(* IEC 61131-3 sources: mect_apps/AnyTPAC/TestSuite/plc, 74 files *)

(* ---- Crosstable.gvl ---- *)
VAR_GLOBAL
	LogLevel AT %QW0.764:INT;
	Target AT %QD0.768:UDINT;
	Status AT %QD0.772:DINT;
	BUTTON_START AT %QX0.776.0:BOOL;
	BUTTON_STOP AT %QX0.780.0:BOOL;
	BUTTON_RESET AT %QX0.784.0:BOOL;
	Tests AT %QD0.788:UDINT;
	Loops AT %QD0.792:UDINT;
	Errors AT %QD0.796:UDINT;
	Elapsed_s AT %QD0.800:UDINT;
	DisabledTests AT %QW0.804:UINT;
	TestingTests AT %QW0.808:UINT;
	PassedTests AT %QW0.812:UINT;
	FailedTests AT %QW0.816:UINT;
	ETMAX_Task00 AT %QD0.840:UDINT;	(* TSK_GetStatistic().ExecMax *)
	ETMAX_Task01 AT %QD0.844:UDINT;	(* TSK_GetStatistic().ExecMax *)
	ETMAX_Task02 AT %QD0.848:UDINT;	(* TSK_GetStatistic().ExecMax *)
	ETMAX_Task03 AT %QD0.852:UDINT;	(* TSK_GetStatistic().ExecMaxfo *)
	ETMAX_Task04 AT %QD0.856:UDINT;	(* TSK_GetStatistic().ExecMax *)
	ETMAX_Task05 AT %QD0.860:UDINT;	(* TSK_GetStatistic().ExecMax *)
	ETMAX_Task06 AT %QD0.864:UDINT;	(* TSK_GetStatistic().ExecMax *)
	ETMAX_Task07 AT %QD0.868:UDINT;	(* TSK_GetStatistic().ExecMax *)
	ETMAX_Task08 AT %QD0.872:UDINT;	(* TSK_GetStatistic().ExecMax *)
	ETMAX_Task09 AT %QD0.876:UDINT;	(* TSK_GetStatistic().ExecMax *)
	ETMAX_Task10 AT %QD0.880:UDINT;	(* TSK_GetStatistic().ExecMax *)
	ETMAX_Task11 AT %QD0.884:UDINT;	(* TSK_GetStatistic().ExecMax *)
	ETMAX_Task12 AT %QD0.888:UDINT;	(* TSK_GetStatistic().ExecMax *)
	ETMAX_Task13 AT %QD0.892:UDINT;	(* TSK_GetStatistic().ExecMax *)
	ETMAX_Task14 AT %QD0.896:UDINT;	(* TSK_GetStatistic().ExecMaxo *)
	ETMAX_Task15 AT %QD0.900:UDINT;	(* TSK_GetStatistic().ExecMax *)
	ETMAX_Task16 AT %QD0.904:UDINT;	(* TSK_GetStatistic().ExecMax *)
	ETMAX_Task17 AT %QD0.908:UDINT;	(* TSK_GetStatistic().ExecMax *)
	ETMAX_Task18 AT %QD0.912:UDINT;	(* TSK_GetStatistic().ExecMax *)
	ETMAX_Task19 AT %QD0.916:UDINT;	(* TaskInfo *)
	ETAVG_Task00 AT %QD0.960:UDINT;	(* TSK_GetStatistic().ExecAverage *)
	ETAVG_Task01 AT %QD0.964:UDINT;	(* TSK_GetStatistic().ExecAverage *)
	ETAVG_Task02 AT %QD0.968:UDINT;	(* TSK_GetStatistic().ExecAverage *)
	ETAVG_Task03 AT %QD0.972:UDINT;	(* TSK_GetStatistic().ExecAverage *)
	ETAVG_Task04 AT %QD0.976:UDINT;	(* TSK_GetStatistic().ExecAverage *)
	ETAVG_Task05 AT %QD0.980:UDINT;	(* TSK_GetStatistic().ExecAverage *)
	ETAVG_Task06 AT %QD0.984:UDINT;	(* TSK_GetStatistic().ExecAverage *)
	ETAVG_Task07 AT %QD0.988:UDINT;	(* TSK_GetStatistic().ExecAverage *)
	ETAVG_Task08 AT %QD0.992:UDINT;	(* TSK_GetStatistic().ExecAverage *)
	ETAVG_Task09 AT %QD0.996:UDINT;	(* TSK_GetStatistic().ExecAverage *)
	ETAVG_Task10 AT %QD0.1000:UDINT;	(* TSK_GetStatistic().ExecAverage *)
	ETAVG_Task11 AT %QD0.1004:UDINT;	(* TSK_GetStatistic().ExecAverage *)
	ETAVG_Task12 AT %QD0.1008:UDINT;	(* TSK_GetStatistic().ExecAverage *)
	ETAVG_Task13 AT %QD0.1012:UDINT;	(* TSK_GetStatistic().ExecAverage *)
	ETAVG_Task14 AT %QD0.1016:UDINT;	(* TSK_GetStatistic().ExecAverage *)
	ETAVG_Task15 AT %QD0.1020:UDINT;	(* TSK_GetStatistic().ExecAverage *)
	ETAVG_Task16 AT %QD0.1024:UDINT;	(* TSK_GetStatistic().ExecAverage *)
	ETAVG_Task17 AT %QD0.1028:UDINT;	(* TSK_GetStatistic().ExecAverage *)
	ETAVG_Task18 AT %QD0.1032:UDINT;	(* TSK_GetStatistic().ExecAverage *)
	ETAVG_Task19 AT %QD0.1036:UDINT;	(* TSK_GetStatistic().ExecAverage *)
	test_level_01 AT %QW0.1204:UINT;
	test_level_02 AT %QW0.1208:UINT;
	test_level_03 AT %QW0.1212:UINT;
	test_level_04 AT %QW0.1216:UINT;
	test_level_05 AT %QW0.1220:UINT;
	test_level_06 AT %QW0.1224:UINT;
	test_level_07 AT %QW0.1228:UINT;
	test_level_08 AT %QW0.1232:UINT;
	test_level_09 AT %QW0.1236:UINT;
	test_level_10 AT %QW0.1240:UINT;
	test_level_11 AT %QW0.1244:UINT;
	test_level_12 AT %QW0.1248:UINT;
	test_level_13 AT %QW0.1252:UINT;
	test_level_14 AT %QW0.1256:UINT;
	test_level_15 AT %QW0.1260:UINT;
	test_level_16 AT %QW0.1264:UINT;
	test_level_17 AT %QW0.1268:UINT;
	test_level_18 AT %QW0.1272:UINT;
	test_level_19 AT %QW0.1276:UINT;
	test_level_20 AT %QW0.1280:UINT;
	test_level_21 AT %QW0.1284:UINT;
	test_level_22 AT %QW0.1288:UINT;
	test_level_23 AT %QW0.1292:UINT;
	test_level_24 AT %QW0.1296:UINT;
	test_level_25 AT %QW0.1300:UINT;
	test_level_26 AT %QW0.1304:UINT;
	test_level_27 AT %QW0.1308:UINT;
	test_level_28 AT %QW0.1312:UINT;
	test_level_29 AT %QW0.1316:UINT;
	test_level_30 AT %QW0.1320:UINT;
	test_level_31 AT %QW0.1324:UINT;
	test_level_32 AT %QW0.1328:UINT;
	test_level_33 AT %QW0.1332:UINT;
	test_level_34 AT %QW0.1336:UINT;
	test_level_35 AT %QW0.1340:UINT;
	test_level_36 AT %QW0.1344:UINT;
	test_level_37 AT %QW0.1348:UINT;
	test_level_38 AT %QW0.1352:UINT;
	test_level_39 AT %QW0.1356:UINT;
	test_level_40 AT %QW0.1360:UINT;
	test_level_41 AT %QW0.1364:UINT;
	test_level_42 AT %QW0.1368:UINT;
	test_level_43 AT %QW0.1372:UINT;
	test_level_44 AT %QW0.1376:UINT;
	test_level_45 AT %QW0.1380:UINT;
	test_level_46 AT %QW0.1384:UINT;
	test_level_47 AT %QW0.1388:UINT;
	test_level_48 AT %QW0.1392:UINT;
	test_level_49 AT %QW0.1396:UINT;
	test_level_50 AT %QW0.1400:UINT;
	test_level_51 AT %QW0.1404:UINT;
	test_level_52 AT %QW0.1408:UINT;
	test_level_53 AT %QW0.1412:UINT;
	test_level_54 AT %QW0.1416:UINT;
	test_level_55 AT %QW0.1420:UINT;
	test_level_56 AT %QW0.1424:UINT;
	test_level_57 AT %QW0.1428:UINT;
	test_level_58 AT %QW0.1432:UINT;
	test_level_59 AT %QW0.1436:UINT;
	test_level_60 AT %QW0.1440:UINT;
	test_counter_01 AT %QD0.1604:UDINT;
	test_counter_02 AT %QD0.1608:UDINT;
	test_counter_03 AT %QD0.1612:UDINT;
	test_counter_04 AT %QD0.1616:UDINT;
	test_counter_05 AT %QD0.1620:UDINT;
	test_counter_06 AT %QD0.1624:UDINT;
	test_counter_07 AT %QD0.1628:UDINT;
	test_counter_08 AT %QD0.1632:UDINT;
	test_counter_09 AT %QD0.1636:UDINT;
	test_counter_10 AT %QD0.1640:UDINT;
	test_counter_11 AT %QD0.1644:UDINT;
	test_counter_12 AT %QD0.1648:UDINT;
	test_counter_13 AT %QD0.1652:UDINT;
	test_counter_14 AT %QD0.1656:UDINT;
	test_counter_15 AT %QD0.1660:UDINT;
	test_counter_16 AT %QD0.1664:UDINT;
	test_counter_17 AT %QD0.1668:UDINT;
	test_counter_18 AT %QD0.1672:UDINT;
	test_counter_19 AT %QD0.1676:UDINT;
	test_counter_20 AT %QD0.1680:UDINT;
	test_counter_21 AT %QD0.1684:UDINT;
	test_counter_22 AT %QD0.1688:UDINT;
	test_counter_23 AT %QD0.1692:UDINT;
	test_counter_24 AT %QD0.1696:UDINT;
	test_counter_25 AT %QD0.1700:UDINT;
	test_counter_26 AT %QD0.1704:UDINT;
	test_counter_27 AT %QD0.1708:UDINT;
	test_counter_28 AT %QD0.1712:UDINT;
	test_counter_29 AT %QD0.1716:UDINT;
	test_counter_30 AT %QD0.1720:UDINT;
	test_counter_31 AT %QD0.1724:UDINT;
	test_counter_32 AT %QD0.1728:UDINT;
	test_counter_33 AT %QD0.1732:UDINT;
	test_counter_34 AT %QD0.1736:UDINT;
	test_counter_35 AT %QD0.1740:UDINT;
	test_counter_36 AT %QD0.1744:UDINT;
	test_counter_37 AT %QD0.1748:UDINT;
	test_counter_38 AT %QD0.1752:UDINT;
	test_counter_39 AT %QD0.1756:UDINT;
	test_counter_40 AT %QD0.1760:UDINT;
	test_counter_41 AT %QD0.1764:UDINT;
	test_counter_42 AT %QD0.1768:UDINT;
	test_counter_43 AT %QD0.1772:UDINT;
	test_counter_44 AT %QD0.1776:UDINT;
	test_counter_45 AT %QD0.1780:UDINT;
	test_counter_46 AT %QD0.1784:UDINT;
	test_counter_47 AT %QD0.1788:UDINT;
	test_counter_48 AT %QD0.1792:UDINT;
	test_counter_49 AT %QD0.1796:UDINT;
	test_counter_50 AT %QD0.1800:UDINT;
	test_counter_51 AT %QD0.1804:UDINT;
	test_counter_52 AT %QD0.1808:UDINT;
	test_counter_53 AT %QD0.1812:UDINT;
	test_counter_54 AT %QD0.1816:UDINT;
	test_counter_55 AT %QD0.1820:UDINT;
	test_counter_56 AT %QD0.1824:UDINT;
	test_counter_57 AT %QD0.1828:UDINT;
	test_counter_58 AT %QD0.1832:UDINT;
	test_counter_59 AT %QD0.1836:UDINT;
	test_counter_60 AT %QD0.1840:UDINT;
	test_loops_01 AT %QD0.2004:UDINT;
	test_loops_02 AT %QD0.2008:UDINT;
	test_loops_03 AT %QD0.2012:UDINT;
	test_loops_04 AT %QD0.2016:UDINT;
	test_loops_05 AT %QD0.2020:UDINT;
	test_loops_06 AT %QD0.2024:UDINT;
	test_loops_07 AT %QD0.2028:UDINT;
	test_loops_08 AT %QD0.2032:UDINT;
	test_loops_09 AT %QD0.2036:UDINT;
	test_loops_10 AT %QD0.2040:UDINT;
	test_loops_11 AT %QD0.2044:UDINT;
	test_loops_12 AT %QD0.2048:UDINT;
	test_loops_13 AT %QD0.2052:UDINT;
	test_loops_14 AT %QD0.2056:UDINT;
	test_loops_15 AT %QD0.2060:UDINT;
	test_loops_16 AT %QD0.2064:UDINT;
	test_loops_17 AT %QD0.2068:UDINT;
	test_loops_18 AT %QD0.2072:UDINT;
	test_loops_19 AT %QD0.2076:UDINT;
	test_loops_20 AT %QD0.2080:UDINT;
	test_loops_21 AT %QD0.2084:UDINT;
	test_loops_22 AT %QD0.2088:UDINT;
	test_loops_23 AT %QD0.2092:UDINT;
	test_loops_24 AT %QD0.2096:UDINT;
	test_loops_25 AT %QD0.2100:UDINT;
	test_loops_26 AT %QD0.2104:UDINT;
	test_loops_27 AT %QD0.2108:UDINT;
	test_loops_28 AT %QD0.2112:UDINT;
	test_loops_29 AT %QD0.2116:UDINT;
	test_loops_30 AT %QD0.2120:UDINT;
	test_loops_31 AT %QD0.2124:UDINT;
	test_loops_32 AT %QD0.2128:UDINT;
	test_loops_33 AT %QD0.2132:UDINT;
	test_loops_34 AT %QD0.2136:UDINT;
	test_loops_35 AT %QD0.2140:UDINT;
	test_loops_36 AT %QD0.2144:UDINT;
	test_loops_37 AT %QD0.2148:UDINT;
	test_loops_38 AT %QD0.2152:UDINT;
	test_loops_39 AT %QD0.2156:UDINT;
	test_loops_40 AT %QD0.2160:UDINT;
	test_loops_41 AT %QD0.2164:UDINT;
	test_loops_42 AT %QD0.2168:UDINT;
	test_loops_43 AT %QD0.2172:UDINT;
	test_loops_44 AT %QD0.2176:UDINT;
	test_loops_45 AT %QD0.2180:UDINT;
	test_loops_46 AT %QD0.2184:UDINT;
	test_loops_47 AT %QD0.2188:UDINT;
	test_loops_48 AT %QD0.2192:UDINT;
	test_loops_49 AT %QD0.2196:UDINT;
	test_loops_50 AT %QD0.2200:UDINT;
	test_loops_51 AT %QD0.2204:UDINT;
	test_loops_52 AT %QD0.2208:UDINT;
	test_loops_53 AT %QD0.2212:UDINT;
	test_loops_54 AT %QD0.2216:UDINT;
	test_loops_55 AT %QD0.2220:UDINT;
	test_loops_56 AT %QD0.2224:UDINT;
	test_loops_57 AT %QD0.2228:UDINT;
	test_loops_58 AT %QD0.2232:UDINT;
	test_loops_59 AT %QD0.2236:UDINT;
	test_loops_60 AT %QD0.2240:UDINT;
	test_errors_01 AT %QD0.2404:UDINT;
	test_errors_02 AT %QD0.2408:UDINT;
	test_errors_03 AT %QD0.2412:UDINT;
	test_errors_04 AT %QD0.2416:UDINT;
	test_errors_05 AT %QD0.2420:UDINT;
	test_errors_06 AT %QD0.2424:UDINT;
	test_errors_07 AT %QD0.2428:UDINT;
	test_errors_08 AT %QD0.2432:UDINT;
	test_errors_09 AT %QD0.2436:UDINT;
	test_errors_10 AT %QD0.2440:UDINT;
	test_errors_11 AT %QD0.2444:UDINT;
	test_errors_12 AT %QD0.2448:UDINT;
	test_errors_13 AT %QD0.2452:UDINT;
	test_errors_14 AT %QD0.2456:UDINT;
	test_errors_15 AT %QD0.2460:UDINT;
	test_errors_16 AT %QD0.2464:UDINT;
	test_errors_17 AT %QD0.2468:UDINT;
	test_errors_18 AT %QD0.2472:UDINT;
	test_errors_19 AT %QD0.2476:UDINT;
	test_errors_20 AT %QD0.2480:UDINT;
	test_errors_21 AT %QD0.2484:UDINT;
	test_errors_22 AT %QD0.2488:UDINT;
	test_errors_23 AT %QD0.2492:UDINT;
	test_errors_24 AT %QD0.2496:UDINT;
	test_errors_25 AT %QD0.2500:UDINT;
	test_errors_26 AT %QD0.2504:UDINT;
	test_errors_27 AT %QD0.2508:UDINT;
	test_errors_28 AT %QD0.2512:UDINT;
	test_errors_29 AT %QD0.2516:UDINT;
	test_errors_30 AT %QD0.2520:UDINT;
	test_errors_31 AT %QD0.2524:UDINT;
	test_errors_32 AT %QD0.2528:UDINT;
	test_errors_33 AT %QD0.2532:UDINT;
	test_errors_34 AT %QD0.2536:UDINT;
	test_errors_35 AT %QD0.2540:UDINT;
	test_errors_36 AT %QD0.2544:UDINT;
	test_errors_37 AT %QD0.2548:UDINT;
	test_errors_38 AT %QD0.2552:UDINT;
	test_errors_39 AT %QD0.2556:UDINT;
	test_errors_40 AT %QD0.2560:UDINT;
	test_errors_41 AT %QD0.2564:UDINT;
	test_errors_42 AT %QD0.2568:UDINT;
	test_errors_43 AT %QD0.2572:UDINT;
	test_errors_44 AT %QD0.2576:UDINT;
	test_errors_45 AT %QD0.2580:UDINT;
	test_errors_46 AT %QD0.2584:UDINT;
	test_errors_47 AT %QD0.2588:UDINT;
	test_errors_48 AT %QD0.2592:UDINT;
	test_errors_49 AT %QD0.2596:UDINT;
	test_errors_50 AT %QD0.2600:UDINT;
	test_errors_51 AT %QD0.2604:UDINT;
	test_errors_52 AT %QD0.2608:UDINT;
	test_errors_53 AT %QD0.2612:UDINT;
	test_errors_54 AT %QD0.2616:UDINT;
	test_errors_55 AT %QD0.2620:UDINT;
	test_errors_56 AT %QD0.2624:UDINT;
	test_errors_57 AT %QD0.2628:UDINT;
	test_errors_58 AT %QD0.2632:UDINT;
	test_errors_59 AT %QD0.2636:UDINT;
	test_errors_60 AT %QD0.2640:UDINT;
	RTU0_TYPE_PORT AT %ID0.20000:UDINT;
	RTU0_BAUDRATE AT %ID0.20004:UDINT;
	RTU0_STATUS AT %ID0.20008:UDINT;
	RTU0_READS AT %ID0.20012:UDINT;
	RTU0_WRITES AT %ID0.20016:UDINT;
	RTU0_TIMEOUTS AT %ID0.20020:UDINT;
	RTU0_COMM_ERRORS AT %ID0.20024:UDINT;
	RTU0_LAST_ERROR AT %ID0.20028:UDINT;
	RTU0_WRITE_QUEUE AT %ID0.20032:UDINT;
	RTU0_BUS_LOAD AT %ID0.20036:UDINT;
	RTU1_TYPE_PORT AT %ID0.20040:UDINT;
	RTU1_BAUDRATE AT %ID0.20044:UDINT;
	RTU1_STATUS AT %ID0.20048:UDINT;
	RTU1_READS AT %ID0.20052:UDINT;
	RTU1_WRITES AT %ID0.20056:UDINT;
	RTU1_TIMEOUTS AT %ID0.20060:UDINT;
	RTU1_COMM_ERRORS AT %ID0.20064:UDINT;
	RTU1_LAST_ERROR AT %ID0.20068:UDINT;
	RTU1_WRITE_QUEUE AT %ID0.20072:UDINT;
	RTU1_BUS_LOAD AT %ID0.20076:UDINT;
	RTU3_TYPE_PORT AT %ID0.20080:UDINT;
	RTU3_BAUDRATE AT %ID0.20084:UDINT;
	RTU3_STATUS AT %ID0.20088:UDINT;
	RTU3_READS AT %ID0.20092:UDINT;
	RTU3_WRITES AT %ID0.20096:UDINT;
	RTU3_TIMEOUTS AT %ID0.20100:UDINT;
	RTU3_COMM_ERRORS AT %ID0.20104:UDINT;
	RTU3_LAST_ERROR AT %ID0.20108:UDINT;
	RTU3_WRITE_QUEUE AT %ID0.20112:UDINT;
	RTU3_BUS_LOAD AT %ID0.20116:UDINT;
	CAN0_TYPE_PORT AT %ID0.20120:UDINT;
	CAN0_BAUDRATE AT %ID0.20124:UDINT;
	CAN0_STATUS AT %ID0.20128:UDINT;
	CAN0_READS AT %ID0.20132:UDINT;
	CAN0_WRITES AT %ID0.20136:UDINT;
	CAN0_TIMEOUTS AT %ID0.20140:UDINT;
	CAN0_COMM_ERRORS AT %ID0.20144:UDINT;
	CAN0_LAST_ERROR AT %ID0.20148:UDINT;
	CAN0_WRITE_QUEUE AT %ID0.20152:UDINT;
	CAN0_BUS_LOAD AT %ID0.20156:UDINT;
	CAN1_TYPE_PORT AT %ID0.20160:UDINT;
	CAN1_BAUDRATE AT %ID0.20164:UDINT;
	CAN1_STATUS AT %ID0.20168:UDINT;
	CAN1_READS AT %ID0.20172:UDINT;
	CAN1_WRITES AT %ID0.20176:UDINT;
	CAN1_TIMEOUTS AT %ID0.20180:UDINT;
	CAN1_COMM_ERRORS AT %ID0.20184:UDINT;
	CAN1_LAST_ERROR AT %ID0.20188:UDINT;
	CAN1_WRITE_QUEUE AT %ID0.20192:UDINT;
	CAN1_BUS_LOAD AT %ID0.20196:UDINT;
	TCPS_TYPE_PORT AT %ID0.20200:UDINT;
	TCPS_IP_ADDRESS AT %ID0.20204:UDINT;
	TCPS_STATUS AT %ID0.20208:UDINT;
	TCPS_READS AT %ID0.20212:UDINT;
	TCPS_WRITES AT %ID0.20216:UDINT;
	TCPS_TIMEOUTS AT %ID0.20220:UDINT;
	TCPS_COMM_ERRORS AT %ID0.20224:UDINT;
	TCPS_LAST_ERROR AT %ID0.20228:UDINT;
	TCPS_WRITE_QUEUE AT %ID0.20232:UDINT;
	TCPS_BUS_LOAD AT %ID0.20236:UDINT;
	TCP0_TYPE_PORT AT %ID0.20240:UDINT;
	TCP0_IP_ADDRESS AT %ID0.20244:UDINT;
	TCP0_STATUS AT %ID0.20248:UDINT;
	TCP0_READS AT %ID0.20252:UDINT;
	TCP0_WRITES AT %ID0.20256:UDINT;
	TCP0_TIMEOUTS AT %ID0.20260:UDINT;
	TCP0_COMM_ERRORS AT %ID0.20264:UDINT;
	TCP0_LAST_ERROR AT %ID0.20268:UDINT;
	TCP0_WRITE_QUEUE AT %ID0.20272:UDINT;
	TCP0_BUS_LOAD AT %ID0.20276:UDINT;
	TCP1_TYPE_PORT AT %ID0.20280:UDINT;
	TCP1_IP_ADDRESS AT %ID0.20284:UDINT;
	TCP1_STATUS AT %ID0.20288:UDINT;
	TCP1_READS AT %ID0.20292:UDINT;
	TCP1_WRITES AT %ID0.20296:UDINT;
	TCP1_TIMEOUTS AT %ID0.20300:UDINT;
	TCP1_COMM_ERRORS AT %ID0.20304:UDINT;
	TCP1_LAST_ERROR AT %ID0.20308:UDINT;
	TCP1_WRITE_QUEUE AT %ID0.20312:UDINT;
	TCP1_BUS_LOAD AT %ID0.20316:UDINT;
	TCP2_TYPE_PORT AT %ID0.20320:UDINT;
	TCP2_IP_ADDRESS AT %ID0.20324:UDINT;
	TCP2_STATUS AT %ID0.20328:UDINT;
	TCP2_READS AT %ID0.20332:UDINT;
	TCP2_WRITES AT %ID0.20336:UDINT;
	TCP2_TIMEOUTS AT %ID0.20340:UDINT;
	TCP2_COMM_ERRORS AT %ID0.20344:UDINT;
	TCP2_LAST_ERROR AT %ID0.20348:UDINT;
	TCP2_WRITE_QUEUE AT %ID0.20352:UDINT;
	TCP2_BUS_LOAD AT %ID0.20356:UDINT;
	TCP3_TYPE_PORT AT %ID0.20360:UDINT;
	TCP3_IP_ADDRESS AT %ID0.20364:UDINT;
	TCP3_STATUS AT %ID0.20368:UDINT;
	TCP3_READS AT %ID0.20372:UDINT;
	TCP3_WRITES AT %ID0.20376:UDINT;
	TCP3_TIMEOUTS AT %ID0.20380:UDINT;
	TCP3_COMM_ERRORS AT %ID0.20384:UDINT;
	TCP3_LAST_ERROR AT %ID0.20388:UDINT;
	TCP3_WRITE_QUEUE AT %ID0.20392:UDINT;
	TCP3_BUS_LOAD AT %ID0.20396:UDINT;
	TCP4_TYPE_PORT AT %ID0.20400:UDINT;
	TCP4_IP_ADDRESS AT %ID0.20404:UDINT;
	TCP4_STATUS AT %ID0.20408:UDINT;
	TCP4_READS AT %ID0.20412:UDINT;
	TCP4_WRITES AT %ID0.20416:UDINT;
	TCP4_TIMEOUTS AT %ID0.20420:UDINT;
	TCP4_COMM_ERRORS AT %ID0.20424:UDINT;
	TCP4_LAST_ERROR AT %ID0.20428:UDINT;
	TCP4_WRITE_QUEUE AT %ID0.20432:UDINT;
	TCP4_BUS_LOAD AT %ID0.20436:UDINT;
	TCP5_TYPE_PORT AT %ID0.20440:UDINT;
	TCP5_IP_ADDRESS AT %ID0.20444:UDINT;
	TCP5_STATUS AT %ID0.20448:UDINT;
	TCP5_READS AT %ID0.20452:UDINT;
	TCP5_WRITES AT %ID0.20456:UDINT;
	TCP5_TIMEOUTS AT %ID0.20460:UDINT;
	TCP5_COMM_ERRORS AT %ID0.20464:UDINT;
	TCP5_LAST_ERROR AT %ID0.20468:UDINT;
	TCP5_WRITE_QUEUE AT %ID0.20472:UDINT;
	TCP5_BUS_LOAD AT %ID0.20476:UDINT;
	TCP6_TYPE_PORT AT %ID0.20480:UDINT;
	TCP6_IP_ADDRESS AT %ID0.20484:UDINT;
	TCP6_STATUS AT %ID0.20488:UDINT;
	TCP6_READS AT %ID0.20492:UDINT;
	TCP6_WRITES AT %ID0.20496:UDINT;
	TCP6_TIMEOUTS AT %ID0.20500:UDINT;
	TCP6_COMM_ERRORS AT %ID0.20504:UDINT;
	TCP6_LAST_ERROR AT %ID0.20508:UDINT;
	TCP6_WRITE_QUEUE AT %ID0.20512:UDINT;
	TCP6_BUS_LOAD AT %ID0.20516:UDINT;
	TCP7_TYPE_PORT AT %ID0.20520:UDINT;
	TCP7_IP_ADDRESS AT %ID0.20524:UDINT;
	TCP7_STATUS AT %ID0.20528:UDINT;
	TCP7_READS AT %ID0.20532:UDINT;
	TCP7_WRITES AT %ID0.20536:UDINT;
	TCP7_TIMEOUTS AT %ID0.20540:UDINT;
	TCP7_COMM_ERRORS AT %ID0.20544:UDINT;
	TCP7_LAST_ERROR AT %ID0.20548:UDINT;
	TCP7_WRITE_QUEUE AT %ID0.20552:UDINT;
	TCP7_BUS_LOAD AT %ID0.20556:UDINT;
	TCP8_TYPE_PORT AT %ID0.20560:UDINT;
	TCP8_IP_ADDRESS AT %ID0.20564:UDINT;
	TCP8_STATUS AT %ID0.20568:UDINT;
	TCP8_READS AT %ID0.20572:UDINT;
	TCP8_WRITES AT %ID0.20576:UDINT;
	TCP8_TIMEOUTS AT %ID0.20580:UDINT;
	TCP8_COMM_ERRORS AT %ID0.20584:UDINT;
	TCP8_LAST_ERROR AT %ID0.20588:UDINT;
	TCP8_WRITE_QUEUE AT %ID0.20592:UDINT;
	TCP8_BUS_LOAD AT %ID0.20596:UDINT;
	TCP9_TYPE_PORT AT %ID0.20600:UDINT;
	TCP9_IP_ADDRESS AT %ID0.20604:UDINT;
	TCP9_STATUS AT %ID0.20608:UDINT;
	TCP9_READS AT %ID0.20612:UDINT;
	TCP9_WRITES AT %ID0.20616:UDINT;
	TCP9_TIMEOUTS AT %ID0.20620:UDINT;
	TCP9_COMM_ERRORS AT %ID0.20624:UDINT;
	TCP9_LAST_ERROR AT %ID0.20628:UDINT;
	TCP9_WRITE_QUEUE AT %ID0.20632:UDINT;
	TCP9_BUS_LOAD AT %ID0.20636:UDINT;
	NODE_01_DEV_NODE AT %ID0.20688:UDINT;
	NODE_01_STATUS AT %ID0.20692:UDINT;
	NODE_02_DEV_NODE AT %ID0.20696:UDINT;
	NODE_02_STATUS AT %ID0.20700:UDINT;
	NODE_03_DEV_NODE AT %ID0.20704:UDINT;
	NODE_03_STATUS AT %ID0.20708:UDINT;
	NODE_04_DEV_NODE AT %ID0.20712:UDINT;
	NODE_04_STATUS AT %ID0.20716:UDINT;
	NODE_05_DEV_NODE AT %ID0.20720:UDINT;
	NODE_05_STATUS AT %ID0.20724:UDINT;
	NODE_06_DEV_NODE AT %ID0.20728:UDINT;
	NODE_06_STATUS AT %ID0.20732:UDINT;
	NODE_07_DEV_NODE AT %ID0.20736:UDINT;
	NODE_07_STATUS AT %ID0.20740:UDINT;
	NODE_08_DEV_NODE AT %ID0.20744:UDINT;
	NODE_08_STATUS AT %ID0.20748:UDINT;
	NODE_09_DEV_NODE AT %ID0.20752:UDINT;
	NODE_09_STATUS AT %ID0.20756:UDINT;
	NODE_10_DEV_NODE AT %ID0.20760:UDINT;
	NODE_10_STATUS AT %ID0.20764:UDINT;
	NODE_11_DEV_NODE AT %ID0.20768:UDINT;
	NODE_11_STATUS AT %ID0.20772:UDINT;
	NODE_12_DEV_NODE AT %ID0.20776:UDINT;
	NODE_12_STATUS AT %ID0.20780:UDINT;
	NODE_13_DEV_NODE AT %ID0.20784:UDINT;
	NODE_13_STATUS AT %ID0.20788:UDINT;
	NODE_14_DEV_NODE AT %ID0.20792:UDINT;
	NODE_14_STATUS AT %ID0.20796:UDINT;
	NODE_15_DEV_NODE AT %ID0.20800:UDINT;
	NODE_15_STATUS AT %ID0.20804:UDINT;
	NODE_16_DEV_NODE AT %ID0.20808:UDINT;
	NODE_16_STATUS AT %ID0.20812:UDINT;
	PLC_time AT %ID0.21560:REAL;	(* Seconds since boot (reset each 24h) *)
	PLC_timeMin AT %ID0.21564:REAL;	(* 10 seconds window start *)
	PLC_timeMax AT %ID0.21568:REAL;	(* 10 seconds window stop *)
	PLC_timeWin AT %QD0.21572:REAL;	(* Graph display window *)
	PLC_Version AT %IW0.21576:UINT;	(* Run Time version *)
	PLC_EngineStatus AT %IW0.21580:UINT;	(* PLC status *)
	PLC_ResetValues AT %QX0.21584.0:BOOL;	(* Diagnostic variables reset *)
	PLC_buzzerOn AT %QX0.21588.0:BOOL;	(* Buzzer sound (enable = 1 disable = 0) *)
	PLC_PLC_Version AT %QW0.21592:UINT;	(* PLC application version *)
	PLC_HMI_Version AT %QW0.21596:UINT;	(* HMI application version *)
	PLC_Year AT %IW0.21640:UINT;	(* Currently year *)
	PLC_Month AT %IW0.21644:UINT;	(* Currently month *)
	PLC_Day AT %IW0.21648:UINT;	(* Currently day *)
	PLC_Hours AT %IW0.21652:UINT;	(* Currently hour *)
	PLC_Minutes AT %IW0.21656:UINT;	(* Currently minutes *)
	PLC_Seconds AT %IW0.21660:UINT;	(* Currently seconds *)
	PLC_UPTIME_s AT %ID0.21664:UDINT;	(* Uptime in seconds (wraps in 136 years) *)
	PLC_UPTIME_cs AT %ID0.21668:UDINT;	(* Uptime in centiseconds = 10 ms (wraps in 497 days) *)
	PLC_WATCHDOGEN AT %QX0.21672.0:BOOL;	(* Enable Watchdog *)
	PLC_WATCHDOG_ms AT %QD0.21676:UDINT;	(* Reset Watchdog timer *)
	PLC_PRODUCT_ID AT %ID0.21680:UDINT;	(* TP/TPAC/TPLC Product ID (Hex) *)
	PLC_SERIAL_NUMBER AT %ID0.21684:UDINT;	(* TP/TPAC/TPLC Serial Number *)
	PLC_HMI_PAGE AT %QD0.21688:DINT;	(* HMI Page (page100=0x00000100) *)
	PLC_BEEP_VOLUME AT %QB0.21740:BYTE;	(* Beep volume (when buzzerOn) *)
	PLC_TOUCH_VOLUME AT %QB0.21744:BYTE;	(* Touch volume *)
	PLC_ALARM_VOLUME AT %QB0.21748:BYTE;	(* Alarm volume (when alarm) *)
	PLC_BUZZER AT %QD0.21752:UDINT;	(* Enable dynamic buzzer sound (0x44332211 up=0x11(%) on=0x22(cs) off=0x33(cs) rep=0x44(times)) *)
END_VAR

(* ---- Resource1.gvl ---- *)
(* Global variable file *)

VAR_GLOBAL

	log_file : F_SYNC_FILE;

	test_names : array [1..test_num] of string := [
	(* 01 *) 'ATCM_IEC1131_3:bool_to_*',
	(* 02 *) 'ATCM_IEC1131_3:byte_to_*',
	(* 03 *) 'ATCM_IEC1131_3:dint_to_*',
	(* 04 *) 'ATCM_IEC1131_3:dword_to_*',
	(* 05 *) 'ATCM_IEC1131_3:int_to_*',
	(* 06 *) 'ATCM_IEC1131_3:lreal_to_*',
	(* 07 *) 'ATCM_IEC1131_3:real_to_*',
	(* 08 *) 'ATCM_IEC1131_3:string_to_*',
	(* 09 *) 'ATCM_IEC1131_3:time_to_*',
	(* 10 *) 'ATCM_IEC1131_3:trunc_to_*',
	(* 11 *) 'ATCM_IEC1131_3:udint_to_*',
	(* 12 *) 'ATCM_IEC1131_3:uint_to_*',
	(* 13 *) 'ATCM_IEC1131_3:word_to_*',
	(* 14 *) 'ATCM_IEC1131_3:ABS',
	(* 15 *) 'ATCM_IEC1131_3:TRIG_INV=ASIN+ACOS+ATAN',
	(* 16 *) 'ATCM_IEC1131_3:TRIG=SIN+COS+TAN',
	(* 17 *) 'ATCM_IEC1131_3:POW=EXP+LN+LOG+SQRT',
	(* 18 *) 'ATCM_IEC1131_3:ADD',
	(* 19 *) 'ATCM_IEC1131_3:DIV',
	(* 20 *) 'ATCM_IEC1131_3:EXPT',
	(* 21 *) 'ATCM_IEC1131_3:MOD',
	(* 22 *) 'ATCM_IEC1131_3:MOVE',
	(* 23 *) 'ATCM_IEC1131_3:MUL',
	(* 24 *) 'ATCM_IEC1131_3:SUB',
	(* 25 *) 'ATCM_IEC1131_3:RO=ROL+ROR',
	(* 26 *) 'ATCM_IEC1131_3:SH=SHL+SHR',
	(* 27 *) 'ATCM_IEC1131_3:AND',
	(* 28 *) 'ATCM_IEC1131_3:NOT',
	(* 29 *) 'ATCM_IEC1131_3:OR',
	(* 30 *) 'ATCM_IEC1131_3:XOR',
	(* 31 *) 'ATCM_IEC1131_3:LIMIT',
	(* 32 *) 'ATCM_IEC1131_3:MAX',
	(* 33 *) 'ATCM_IEC1131_3:MIN',
	(* 34 *) 'ATCM_IEC1131_3:MUX',
	(* 35 *) 'ATCM_IEC1131_3:SEL',
	(* 36 *) 'ATCM_IEC1131_3:EQ',
	(* 37 *) 'ATCM_IEC1131_3:GE',
	(* 38 *) 'ATCM_IEC1131_3:GT',
	(* 39 *) 'ATCM_IEC1131_3:LE',
	(* 40 *) 'ATCM_IEC1131_3:LT',
	(* 41 *) 'ATCM_IEC1131_3:NE',
	(* 42 *) 'ATCM_IEC1131_3:CONCAT',
	(* 43 *) 'ATCM_IEC1131_3:DELETE',
	(* 44 *) 'ATCM_IEC1131_3:FIND',
	(* 45 *) 'ATCM_IEC1131_3:INSERT',
	(* 46 *) 'ATCM_IEC1131_3:LEFT=LEFT+RIGHT',
	(* 47 *) 'ATCM_IEC1131_3:LEN',
	(* 48 *) 'ATCM_IEC1131_3:MID',
	(* 49 *) 'ATCM_IEC1131_3:REPLACE',
	(* 50 *) 'ATCM_IEC1131_3:ADDTIME+SUBTIME',
	(* 51 *) 'ATCM_IEC1131_3:DIVTIME+MULTIME',
	(* 52 *) 'ATCM_IEC1131_3:RS+SR',
	(* 53 *) 'ATCM_IEC1131_3:F_TRIG+R_TRIG',
	(* 54 *) 'ATCM_IEC1131_3:CTD+CTU+CTUD',
	(* 55 *) 'ATCM_IEC1131_3:TOF+TON+TP',
	(* 56 *) 'ATCM_Utility:BYTE_SWAP_DWORD+WORD',
	(* 57 *) 'ATCM_Utility:COPY_FROM+TO_BYTE_ARRAY',
	(* 58 *) 'ATCM_Utility:HI+LO_BYTE+WORD',
	(* 59 *) 'ATCM_Utility:MAKE_DWORD+WORD',
    (* 60 *) ''
	];

END_VAR

(* ---- ResetCounters.st ---- *)
(*[[
]]*)
FUNCTION ResetCounters
#import "Crosstable.gvl"
#import "Resource1.gvl"
VAR
	retval : WORD;
END_VAR;

	Elapsed_s := 0;
	Loops := 0;
	Errors := 0;

	(* no Task00_TestInit *)
	retval := TSK_ClearStatistic('Task01_TestManager');
	retval := TSK_ClearStatistic('Task02_TestMonitor');

	retval := TSK_ClearStatistic('Task03_ATCM_File');
	retval := TSK_ClearStatistic('Task04_ATCM_IEC1131_3_A');
	retval := TSK_ClearStatistic('Task05_ATCM_IEC1131_3_B');
	retval := TSK_ClearStatistic('Task06_ATCM_IEC1131_3_C');
	retval := TSK_ClearStatistic('Task07_ATCM_IEC1131_3_D');
	retval := TSK_ClearStatistic('Task08_ATCM_IEC1131_3_E');
	retval := TSK_ClearStatistic('Task09_ATCM_IEC1131_3_F');
	retval := TSK_ClearStatistic('Task10_ATCM_IEC1131_3_G');
	retval := TSK_ClearStatistic('Task11_ATCM_IEC1131_3_H');
	retval := TSK_ClearStatistic('Task12_ATCM_IEC1131_3_I');
	retval := TSK_ClearStatistic('Task13_ATCM_IEC1131_3_J');
	retval := TSK_ClearStatistic('Task14_ATCM_IEC1131_3_K');
	retval := TSK_ClearStatistic('Task15_ATCM_IEC1131_3_L');
	retval := TSK_ClearStatistic('Task16_ATCM_IEC1131_3_M');
	retval := TSK_ClearStatistic('Task17_ATCM_System');
	retval := TSK_ClearStatistic('Task18_ATCM_System2');
	retval := TSK_ClearStatistic('Task19_ATCM_Utility');

    test_loops_01 := 0;
    test_loops_02 := 0;
    test_loops_03 := 0;
    test_loops_04 := 0;
    test_loops_05 := 0;
    test_loops_06 := 0;
    test_loops_07 := 0;
    test_loops_08 := 0;
    test_loops_09 := 0;
    test_loops_10 := 0;
    test_loops_11 := 0;
    test_loops_12 := 0;
    test_loops_13 := 0;
    test_loops_14 := 0;
    test_loops_15 := 0;
    test_loops_16 := 0;
    test_loops_17 := 0;
    test_loops_18 := 0;
    test_loops_19 := 0;
    test_loops_20 := 0;
    test_loops_21 := 0;
    test_loops_22 := 0;
    test_loops_23 := 0;
    test_loops_24 := 0;
    test_loops_25 := 0;
    test_loops_26 := 0;
    test_loops_27 := 0;
    test_loops_28 := 0;
    test_loops_29 := 0;
    test_loops_30 := 0;
    test_loops_31 := 0;
    test_loops_32 := 0;
    test_loops_33 := 0;
    test_loops_34 := 0;
    test_loops_35 := 0;
    test_loops_36 := 0;
    test_loops_37 := 0;
    test_loops_38 := 0;
    test_loops_39 := 0;
    test_loops_40 := 0;
    test_loops_41 := 0;
    test_loops_42 := 0;
    test_loops_43 := 0;
    test_loops_44 := 0;
    test_loops_45 := 0;
    test_loops_46 := 0;
    test_loops_47 := 0;
    test_loops_48 := 0;
    test_loops_49 := 0;
    test_loops_50 := 0;
    test_loops_51 := 0;
    test_loops_52 := 0;
    test_loops_53 := 0;
    test_loops_54 := 0;
    test_loops_55 := 0;
    test_loops_56 := 0;
    test_loops_57 := 0;
    test_loops_58 := 0;
    test_loops_59 := 0;
    test_loops_60 := 0;

    test_counter_01 := 0;
    test_counter_02 := 0;
    test_counter_03 := 0;
    test_counter_04 := 0;
    test_counter_05 := 0;
    test_counter_06 := 0;
    test_counter_07 := 0;
    test_counter_08 := 0;
    test_counter_09 := 0;
    test_counter_10 := 0;
    test_counter_11 := 0;
    test_counter_12 := 0;
    test_counter_13 := 0;
    test_counter_14 := 0;
    test_counter_15 := 0;
    test_counter_16 := 0;
    test_counter_17 := 0;
    test_counter_18 := 0;
    test_counter_19 := 0;
    test_counter_20 := 0;
    test_counter_21 := 0;
    test_counter_22 := 0;
    test_counter_23 := 0;
    test_counter_24 := 0;
    test_counter_25 := 0;
    test_counter_26 := 0;
    test_counter_27 := 0;
    test_counter_28 := 0;
    test_counter_29 := 0;
    test_counter_30 := 0;
    test_counter_31 := 0;
    test_counter_32 := 0;
    test_counter_33 := 0;
    test_counter_34 := 0;
    test_counter_35 := 0;
    test_counter_36 := 0;
    test_counter_37 := 0;
    test_counter_38 := 0;
    test_counter_39 := 0;
    test_counter_40 := 0;
    test_counter_41 := 0;
    test_counter_42 := 0;
    test_counter_43 := 0;
    test_counter_44 := 0;
    test_counter_45 := 0;
    test_counter_46 := 0;
    test_counter_47 := 0;
    test_counter_48 := 0;
    test_counter_49 := 0;
    test_counter_50 := 0;
    test_counter_51 := 0;
    test_counter_52 := 0;
    test_counter_53 := 0;
    test_counter_54 := 0;
    test_counter_55 := 0;
    test_counter_56 := 0;
    test_counter_57 := 0;
    test_counter_58 := 0;
    test_counter_59 := 0;
    test_counter_60 := 0;

    test_errors_01 := 0;
    test_errors_02 := 0;
    test_errors_03 := 0;
    test_errors_04 := 0;
    test_errors_05 := 0;
    test_errors_06 := 0;
    test_errors_07 := 0;
    test_errors_08 := 0;
    test_errors_09 := 0;
    test_errors_10 := 0;
    test_errors_11 := 0;
    test_errors_12 := 0;
    test_errors_13 := 0;
    test_errors_14 := 0;
    test_errors_15 := 0;
    test_errors_16 := 0;
    test_errors_17 := 0;
    test_errors_18 := 0;
    test_errors_19 := 0;
    test_errors_20 := 0;
    test_errors_21 := 0;
    test_errors_22 := 0;
    test_errors_23 := 0;
    test_errors_24 := 0;
    test_errors_25 := 0;
    test_errors_26 := 0;
    test_errors_27 := 0;
    test_errors_28 := 0;
    test_errors_29 := 0;
    test_errors_30 := 0;
    test_errors_31 := 0;
    test_errors_32 := 0;
    test_errors_33 := 0;
    test_errors_34 := 0;
    test_errors_35 := 0;
    test_errors_36 := 0;
    test_errors_37 := 0;
    test_errors_38 := 0;
    test_errors_39 := 0;
    test_errors_40 := 0;
    test_errors_41 := 0;
    test_errors_42 := 0;
    test_errors_43 := 0;
    test_errors_44 := 0;
    test_errors_45 := 0;
    test_errors_46 := 0;
    test_errors_47 := 0;
    test_errors_48 := 0;
    test_errors_49 := 0;
    test_errors_50 := 0;
    test_errors_51 := 0;
    test_errors_52 := 0;
    test_errors_53 := 0;
    test_errors_54 := 0;
    test_errors_55 := 0;
    test_errors_56 := 0;
    test_errors_57 := 0;
    test_errors_58 := 0;
    test_errors_59 := 0;
    test_errors_60 := 0;

END_FUNCTION

(* ---- SetCompletedLoops.st ---- *)
(*[[
]]*)
FUNCTION SetCompletedLoops
VAR_INPUT
	test_level : UINT;
	test_loops : UDINT;
END_VAR
VAR_IN_OUT
	first : BOOL;
	completedLoops : UDINT;
END_VAR

	if test_level > TEST_DISABLED then
		if first then
			first := false;
			completedLoops := test_loops;
		elsif test_loops < completedLoops then
			completedLoops := test_loops;
		end_if;
	end_if;

END_FUNCTION

(* ---- SetDefaultValues.st ---- *)
(*[[
]]*)
FUNCTION SetDefaultValues
#import "Crosstable.gvl"
#import "Resource1.gvl"

    test_level_01 := TEST_UNKNOWN;
    test_level_02 := TEST_UNKNOWN;
    test_level_03 := TEST_UNKNOWN;
    test_level_04 := TEST_UNKNOWN;
    test_level_05 := TEST_UNKNOWN;
    test_level_06 := TEST_UNKNOWN;
    test_level_07 := TEST_UNKNOWN;
    test_level_08 := TEST_UNKNOWN;
    test_level_09 := TEST_UNKNOWN;
    test_level_10 := TEST_UNKNOWN;
    test_level_11 := TEST_UNKNOWN;
    test_level_12 := TEST_UNKNOWN;
    test_level_13 := TEST_UNKNOWN;
    test_level_14 := TEST_UNKNOWN;
    test_level_15 := TEST_UNKNOWN;
    test_level_16 := TEST_UNKNOWN;
    test_level_17 := TEST_UNKNOWN;
    test_level_18 := TEST_UNKNOWN;
    test_level_19 := TEST_UNKNOWN;
    test_level_20 := TEST_UNKNOWN;
    test_level_21 := TEST_UNKNOWN;
    test_level_22 := TEST_UNKNOWN;
    test_level_23 := TEST_UNKNOWN;
    test_level_24 := TEST_UNKNOWN;
    test_level_25 := TEST_UNKNOWN;
    test_level_26 := TEST_UNKNOWN;
    test_level_27 := TEST_UNKNOWN;
    test_level_28 := TEST_UNKNOWN;
    test_level_29 := TEST_UNKNOWN;
    test_level_30 := TEST_UNKNOWN;
    test_level_31 := TEST_UNKNOWN;
    test_level_32 := TEST_UNKNOWN;
    test_level_33 := TEST_UNKNOWN;
    test_level_34 := TEST_UNKNOWN;
    test_level_35 := TEST_UNKNOWN;
    test_level_36 := TEST_UNKNOWN;
    test_level_37 := TEST_UNKNOWN;
    test_level_38 := TEST_UNKNOWN;
    test_level_39 := TEST_UNKNOWN;
    test_level_40 := TEST_UNKNOWN;
    test_level_41 := TEST_UNKNOWN;
    test_level_42 := TEST_UNKNOWN;
    test_level_43 := TEST_UNKNOWN;
    test_level_44 := TEST_UNKNOWN;
    test_level_45 := TEST_UNKNOWN;
    test_level_46 := TEST_UNKNOWN;
    test_level_47 := TEST_UNKNOWN;
    test_level_48 := TEST_UNKNOWN;
    test_level_49 := TEST_UNKNOWN;
    test_level_50 := TEST_UNKNOWN;
    test_level_51 := TEST_UNKNOWN;
    test_level_52 := TEST_UNKNOWN;
    test_level_53 := TEST_UNKNOWN;
    test_level_54 := TEST_UNKNOWN;
    test_level_55 := TEST_UNKNOWN;
    test_level_56 := TEST_UNKNOWN;
    test_level_57 := TEST_UNKNOWN;
    test_level_58 := TEST_UNKNOWN;
    test_level_59 := TEST_UNKNOWN;
    test_level_60 := TEST_DISABLED;

END_FUNCTION

(* ---- SingleTest.st ---- *)
(*[[
]]*)
FUNCTION SingleTest

#import "Crosstable.gvl"
#import "Resource1.gvl"

VAR_INPUT
	test_id : int;
	passed : bool;
	expected : string;
	obtained : string;
	test_cases : int;
END_VAR

VAR_IN_OUT
	test_index : int;
	test_level: UINT;
    test_counter : UDINT;
	test_loops : UDINT;
    test_errors : UDINT;
END_VAR

VAR
	ignored : bool;
	retval : dint;
	header : string;
	newline : string := '$n';
	m : int;
END_VAR

	(* 1/3 updating the test counters *)
	test_counter := test_counter + 1;
	if not passed then
		test_errors := test_errors + 1;
		Errors := Errors + 1;
		if test_level = TEST_UNKNOWN or test_level = TEST_PASSED then
			test_level := TEST_FAILED;
		end_if;
	end_if;

	(* 2/3 logging, if necessary *)
	if (not passed and LogLevel >= LOG_FAILED_TESTS) or (LogLevel = LOG_PASSED_TESTS) then
		header := time_to_string(tim_get());
		header := CONCAT(header, comma_blank, '"', test_names[test_id], '"');
		header := CONCAT(header, comma_blank, int_to_string(test_index));
		if passed then
			header := CONCAT(header, comma_blank, 'PASSED');
		else
			header := CONCAT(header, comma_blank, 'FAILED');
		end_if;

		 (* remember the 255 string len limit *)
		ignored := F_SYNC_WRITEFILE(header,                          log_file);
		ignored := F_SYNC_WRITEFILE(concat(comma_blank, 'expected'), log_file);
		ignored := F_SYNC_WRITEFILE(expected,                        log_file);
		m := len(expected);
		if (m = 255) then
			ignored := F_SYNC_WRITEFILE('<-LEN', log_file);
		end_if;
		ignored := F_SYNC_WRITEFILE(concat(comma_blank, 'obtained'), log_file);
		ignored := F_SYNC_WRITEFILE(obtained,                        log_file);
		m := len(obtained);
		if (m = 255) then
			ignored := F_SYNC_WRITEFILE('<-LEN', log_file);
		end_if;
		ignored := F_SYNC_WRITEFILE(newline,                         log_file);
		retval := F_FLUSH();
	end_if;

	(* 3/3 updating the loop counters *)
	test_index := test_index + 1;
	if (test_index > test_cases) then
		test_index := 1;
		test_loops := test_loops + 1;
		if test_level = TEST_UNKNOWN then
			test_level := TEST_PASSED;
		end_if;
    end_if;

END_FUNCTION

(* ---- StartTest.st ---- *)
(*[[
]]*)
FUNCTION StartTest
#import "Crosstable.gvl"
#import "Resource1.gvl"

	if LogLevel > LOG_NOTHING then
		log_file.filename := concat(
			'/local/root/TestSuite_',
			time_to_string(getTimeSinceSystemBoot()),
			'.csv');
		log_file.mode := CF_READ_WRITE;
		if not F_SYNC_OPENFILE(log_file) then
			(* FIXME: report error *);
		end_if;
	end_if;

	StartLocalTask('Task03_ATCM_File');
	StartLocalTask('Task04_ATCM_IEC1131_3_A');
	StartLocalTask('Task05_ATCM_IEC1131_3_B');
	StartLocalTask('Task06_ATCM_IEC1131_3_C');
	StartLocalTask('Task07_ATCM_IEC1131_3_D');
	StartLocalTask('Task08_ATCM_IEC1131_3_E');
	StartLocalTask('Task09_ATCM_IEC1131_3_F');
	StartLocalTask('Task10_ATCM_IEC1131_3_G');
	StartLocalTask('Task11_ATCM_IEC1131_3_H');
	StartLocalTask('Task12_ATCM_IEC1131_3_I');
	StartLocalTask('Task13_ATCM_IEC1131_3_J');
	StartLocalTask('Task14_ATCM_IEC1131_3_K');
	StartLocalTask('Task15_ATCM_IEC1131_3_L');
	StartLocalTask('Task16_ATCM_IEC1131_3_M');
	StartLocalTask('Task17_ATCM_System');
	StartLocalTask('Task18_ATCM_System2');
	StartLocalTask('Task19_ATCM_Utility');

END_FUNCTION

(* ---- StepTest.st ---- *)
(*[[
]]*)
FUNCTION StepTest
#import "Crosstable.gvl"
#import "Resource1.gvl"

VAR
	first : bool := true;
	completedLoops : UDINT := 0;
END_VAR

	if LogLevel > LOG_NOTHING then
		;
	end_if;

	(* minimun common completed loops *)
	first := true;
	completedLoops := 0;

	SetCompletedLoops(test_level_01, test_loops_01, first, completedLoops);
	SetCompletedLoops(test_level_02, test_loops_02, first, completedLoops);
	SetCompletedLoops(test_level_03, test_loops_03, first, completedLoops);
	SetCompletedLoops(test_level_04, test_loops_04, first, completedLoops);
	SetCompletedLoops(test_level_05, test_loops_05, first, completedLoops);
	SetCompletedLoops(test_level_06, test_loops_06, first, completedLoops);
	SetCompletedLoops(test_level_07, test_loops_07, first, completedLoops);
	SetCompletedLoops(test_level_08, test_loops_08, first, completedLoops);
	SetCompletedLoops(test_level_09, test_loops_09, first, completedLoops);
	SetCompletedLoops(test_level_10, test_loops_10, first, completedLoops);
	SetCompletedLoops(test_level_11, test_loops_11, first, completedLoops);
	SetCompletedLoops(test_level_12, test_loops_12, first, completedLoops);
	SetCompletedLoops(test_level_13, test_loops_13, first, completedLoops);
	SetCompletedLoops(test_level_14, test_loops_14, first, completedLoops);
	SetCompletedLoops(test_level_15, test_loops_15, first, completedLoops);
	SetCompletedLoops(test_level_16, test_loops_16, first, completedLoops);
	SetCompletedLoops(test_level_17, test_loops_17, first, completedLoops);
	SetCompletedLoops(test_level_18, test_loops_18, first, completedLoops);
	SetCompletedLoops(test_level_19, test_loops_19, first, completedLoops);
	SetCompletedLoops(test_level_20, test_loops_20, first, completedLoops);
	SetCompletedLoops(test_level_21, test_loops_21, first, completedLoops);
	SetCompletedLoops(test_level_22, test_loops_22, first, completedLoops);
	SetCompletedLoops(test_level_23, test_loops_23, first, completedLoops);
	SetCompletedLoops(test_level_24, test_loops_24, first, completedLoops);
	SetCompletedLoops(test_level_25, test_loops_25, first, completedLoops);
	SetCompletedLoops(test_level_26, test_loops_26, first, completedLoops);
	SetCompletedLoops(test_level_27, test_loops_27, first, completedLoops);
	SetCompletedLoops(test_level_28, test_loops_28, first, completedLoops);
	SetCompletedLoops(test_level_29, test_loops_29, first, completedLoops);
	SetCompletedLoops(test_level_30, test_loops_30, first, completedLoops);
	SetCompletedLoops(test_level_31, test_loops_31, first, completedLoops);
	SetCompletedLoops(test_level_32, test_loops_32, first, completedLoops);
	SetCompletedLoops(test_level_33, test_loops_33, first, completedLoops);
	SetCompletedLoops(test_level_34, test_loops_34, first, completedLoops);
	SetCompletedLoops(test_level_35, test_loops_35, first, completedLoops);
	SetCompletedLoops(test_level_36, test_loops_36, first, completedLoops);
	SetCompletedLoops(test_level_37, test_loops_37, first, completedLoops);
	SetCompletedLoops(test_level_38, test_loops_38, first, completedLoops);
	SetCompletedLoops(test_level_39, test_loops_39, first, completedLoops);
	SetCompletedLoops(test_level_40, test_loops_40, first, completedLoops);
	SetCompletedLoops(test_level_41, test_loops_41, first, completedLoops);
	SetCompletedLoops(test_level_42, test_loops_42, first, completedLoops);
	SetCompletedLoops(test_level_43, test_loops_43, first, completedLoops);
	SetCompletedLoops(test_level_44, test_loops_44, first, completedLoops);
	SetCompletedLoops(test_level_45, test_loops_45, first, completedLoops);
	SetCompletedLoops(test_level_46, test_loops_46, first, completedLoops);
	SetCompletedLoops(test_level_47, test_loops_47, first, completedLoops);
	SetCompletedLoops(test_level_48, test_loops_48, first, completedLoops);
	SetCompletedLoops(test_level_49, test_loops_49, first, completedLoops);
	SetCompletedLoops(test_level_50, test_loops_50, first, completedLoops);
	SetCompletedLoops(test_level_51, test_loops_51, first, completedLoops);
	SetCompletedLoops(test_level_52, test_loops_52, first, completedLoops);
	SetCompletedLoops(test_level_53, test_loops_53, first, completedLoops);
	SetCompletedLoops(test_level_54, test_loops_54, first, completedLoops);
	SetCompletedLoops(test_level_55, test_loops_55, first, completedLoops);
	SetCompletedLoops(test_level_56, test_loops_56, first, completedLoops);
	SetCompletedLoops(test_level_57, test_loops_57, first, completedLoops);
	SetCompletedLoops(test_level_58, test_loops_58, first, completedLoops);
	SetCompletedLoops(test_level_59, test_loops_59, first, completedLoops);
	SetCompletedLoops(test_level_60, test_loops_60, first, completedLoops);

	Loops := completedLoops;

END_FUNCTION

(* ---- StopTest.st ---- *)
(*[[
]]*)
FUNCTION StopTest
#import "Crosstable.gvl"
#import "Resource1.gvl"

	StopLocalTask('Task03_ATCM_File');
	StopLocalTask('Task04_ATCM_IEC1131_3_A');
	StopLocalTask('Task05_ATCM_IEC1131_3_B');
	StopLocalTask('Task06_ATCM_IEC1131_3_C');
	StopLocalTask('Task07_ATCM_IEC1131_3_D');
	StopLocalTask('Task08_ATCM_IEC1131_3_E');
	StopLocalTask('Task09_ATCM_IEC1131_3_F');
	StopLocalTask('Task10_ATCM_IEC1131_3_G');
	StopLocalTask('Task11_ATCM_IEC1131_3_H');
	StopLocalTask('Task12_ATCM_IEC1131_3_I');
	StopLocalTask('Task13_ATCM_IEC1131_3_J');
	StopLocalTask('Task14_ATCM_IEC1131_3_K');
	StopLocalTask('Task15_ATCM_IEC1131_3_L');
	StopLocalTask('Task16_ATCM_IEC1131_3_M');
	StopLocalTask('Task17_ATCM_System');
	StopLocalTask('Task18_ATCM_System2');
	StopLocalTask('Task19_ATCM_Utility');

	if LogLevel > LOG_NOTHING then
		if not F_SYNC_CLOSEFILE(log_file) then
			(* FIXME: report error *);
		end_if;
	end_if;

END_FUNCTION

(* ---- UpdateCounters.st ---- *)
(*[[
]]*)
FUNCTION UpdateCounters
#import "Crosstable.gvl"
#import "Resource1.gvl"

	DisabledTests := 0;
	TestingTests := 0;
	PassedTests := 0;
	FailedTests := 0;

    UpdateCountersN(test_level_01);
    UpdateCountersN(test_level_02);
    UpdateCountersN(test_level_03);
    UpdateCountersN(test_level_04);
    UpdateCountersN(test_level_05);
    UpdateCountersN(test_level_06);
    UpdateCountersN(test_level_07);
    UpdateCountersN(test_level_08);
    UpdateCountersN(test_level_09);
    UpdateCountersN(test_level_10);
    UpdateCountersN(test_level_11);
    UpdateCountersN(test_level_12);
    UpdateCountersN(test_level_13);
    UpdateCountersN(test_level_14);
    UpdateCountersN(test_level_15);
    UpdateCountersN(test_level_16);
    UpdateCountersN(test_level_17);
    UpdateCountersN(test_level_18);
    UpdateCountersN(test_level_19);
    UpdateCountersN(test_level_20);
    UpdateCountersN(test_level_21);
    UpdateCountersN(test_level_22);
    UpdateCountersN(test_level_23);
    UpdateCountersN(test_level_24);
    UpdateCountersN(test_level_25);
    UpdateCountersN(test_level_26);
    UpdateCountersN(test_level_27);
    UpdateCountersN(test_level_28);
    UpdateCountersN(test_level_29);
    UpdateCountersN(test_level_30);
    UpdateCountersN(test_level_31);
    UpdateCountersN(test_level_32);
    UpdateCountersN(test_level_33);
    UpdateCountersN(test_level_34);
    UpdateCountersN(test_level_35);
    UpdateCountersN(test_level_36);
    UpdateCountersN(test_level_37);
    UpdateCountersN(test_level_38);
    UpdateCountersN(test_level_39);
    UpdateCountersN(test_level_40);
    UpdateCountersN(test_level_41);
    UpdateCountersN(test_level_42);
    UpdateCountersN(test_level_43);
    UpdateCountersN(test_level_44);
    UpdateCountersN(test_level_45);
    UpdateCountersN(test_level_46);
    UpdateCountersN(test_level_47);
    UpdateCountersN(test_level_48);
    UpdateCountersN(test_level_49);
    UpdateCountersN(test_level_50);
    UpdateCountersN(test_level_51);
    UpdateCountersN(test_level_52);
    UpdateCountersN(test_level_53);
    UpdateCountersN(test_level_54);
    UpdateCountersN(test_level_55);
    UpdateCountersN(test_level_56);
    UpdateCountersN(test_level_57);
    UpdateCountersN(test_level_58);
    UpdateCountersN(test_level_59);
    UpdateCountersN(test_level_60);

END_FUNCTION

(* ---- UpdateCountersN.st ---- *)
(*[[
]]*)
FUNCTION UpdateCountersN
#import "Crosstable.gvl"
#import "Resource1.gvl"
VAR_INPUT
	test_level_N : UINT;
END_VAR

	CASE test_level_N OF
	TEST_DISABLED:
		DisabledTests := DisabledTests + 1;
	TEST_UNKNOWN:
		TestingTests := TestingTests + 1;
	TEST_PASSED:
		PassedTests := PassedTests + 1;
	TEST_FAILED:
		FailedTests := FailedTests + 1;
	ELSE
    	;
    END_CASE;
END_FUNCTION

(* ---- abs_P.st ---- *)
(*[[
]]*)
PROGRAM abs_P
#import "Crosstable.gvl"
#import "Resource1.gvl"
CONST
	this : int := 14;
	test_cases : int := 3;
END_CONST
VAR
	test_case : array [1..test_cases] of lreal_any_num_T :=
[
(input:=-3.1415926535897931, ret_dint:= 3, ret_int:= 3, ret_lreal:= 3.1415926535897931, ret_real:= 3.1415926535897931),
(input:= 0.0000000000000000, ret_dint:= 0, ret_int:= 0, ret_lreal:= 0.0000000000000000, ret_real:= 0.0000000000000000),
(input:= 3.1415926535897931, ret_dint:= 3, ret_int:= 3, ret_lreal:= 3.1415926535897931, ret_real:= 3.1415926535897931)
];
	input_dint ,ret_dint   : dint;
	input_int  ,ret_int    : int;
	input_lreal,ret_lreal  : lreal;
	input_real ,ret_real   : real;
(*
    error C1546: type mismatch: parameter 1 of 'ABS' needs type 'ANY_NUM' but actual is 'BYTE'
    error C1546: type mismatch: parameter 1 of 'ABS' needs type 'ANY_NUM' but actual is 'DWORD'
    error C1562: no implementation found for function overload 'UDINT ABS(UDINT)'
    error C1562: no implementation found for function overload 'UINT ABS(UINT)'
    error C1546: type mismatch: parameter 1 of 'ABS' needs type 'ANY_NUM' but actual is 'WORD'
*)

	index : int := 1;
	expected : string;
	obtained : string;
	result : bool;
END_VAR

	if Status = STATUS_RUNNING AND test_level_14 > TEST_DISABLED and test_loops_14 < Target then

		(* ---------- test action ---------------*)
		input_dint  := lreal_to_dint (test_case[index].input);
		input_int   := lreal_to_int  (test_case[index].input);
		input_lreal := test_case[index].input;
		input_real  := lreal_to_real (test_case[index].input);

		ret_dint  := abs(input_dint );
		ret_int   := abs(input_int  );
		ret_lreal := abs(input_lreal);
		ret_real  := abs(input_real );

		(* ---------- test condition ---------------*)
		result := (ret_dint  = test_case[index].ret_dint )
		      and (ret_int   = test_case[index].ret_int  )
		      and (ret_lreal = test_case[index].ret_lreal)
		      and (ret_real  = test_case[index].ret_real );

		(* ---------- log message ---------------*)
		expected := '';
		expected := CONCAT(expected, comma_blank, dint_to_string(test_case[index].ret_dint ));
		expected := CONCAT(expected, comma_blank, int_to_string(test_case[index].ret_int  ));
		expected := CONCAT(expected, comma_blank, lreal_to_string(test_case[index].ret_lreal));
		expected := CONCAT(expected, comma_blank, real_to_string(test_case[index].ret_real ));
		obtained := '';
		obtained := CONCAT(expected, comma_blank, dint_to_string(ret_dint ));
		obtained := CONCAT(expected, comma_blank, int_to_string(ret_int  ));
		obtained := CONCAT(expected, comma_blank, lreal_to_string(ret_lreal));
		obtained := CONCAT(expected, comma_blank, real_to_string(ret_real ));

		(* ---------- cycle ----------*)
		SingleTest(this, result, expected, obtained, test_cases,
				   index, test_level_14, test_counter_14, test_loops_14, test_errors_14);
	end_if;

END_PROGRAM

(* ---- add_P.st ---- *)
(*[[ ]]*)
PROGRAM add_P
#import "Crosstable.gvl"
#import "Resource1.gvl"
CONST
	this : int := 18;
	test_cases : int := 4;
END_CONST
VAR
	test_case : array [1..test_cases] of num2_num_T := [
		(input0 := 10.0, input1 := 10.0, ret_int := 20, ret_dint := 20, ret_udint := 20, ret_uint := 20, ret_real := 20.0, ret_lreal := 20.0),
		(input0 := 10.0, input1 := 100.0, ret_int := 110, ret_dint := 110, ret_udint := 110, ret_uint := 110, ret_real := 110.0, ret_lreal := 110.0),
		(input0 := -10.0, input1 := 100.0, ret_int := 90, ret_dint := 90, ret_udint := 100, ret_uint := 100, ret_real := 90.0, ret_lreal := 90.0),
		(input0 := -10.0, input1 := -40.0, ret_int := -50, ret_dint := -50, ret_udint := 0, ret_uint := 0, ret_real := -50.0, ret_lreal := -50.0)
	];
    ret_int    : int;
    ret_dint   : dint;
    ret_uint   : uint;
    ret_udint  : udint;
    ret_real   : real;
    ret_lreal  : lreal;

	index : int := 1;
	expected : string;
	obtained : string;
	result : bool;
END_VAR

	if Status = STATUS_RUNNING AND test_level_18 > TEST_DISABLED and test_loops_18 < Target then

		(* ---------- test action ---------------*)
        ret_int     := add(lreal_to_int(test_case[index].input0), lreal_to_int(test_case[index].input1));
        ret_dint    := add(lreal_to_dint(test_case[index].input0), lreal_to_dint(test_case[index].input1));
        ret_uint    := add(lreal_to_uint(test_case[index].input0), lreal_to_uint(test_case[index].input1));
        ret_udint   := add(lreal_to_udint(test_case[index].input0), lreal_to_udint(test_case[index].input1));
        ret_real    := add(lreal_to_real(test_case[index].input0), lreal_to_real(test_case[index].input1));
        ret_lreal   := add(test_case[index].input0, test_case[index].input1);

		(* ---------- test condition ---------------*)
        result := ((ret_int = test_case[index].ret_int)
		      and (ret_dint = test_case[index].ret_dint)
		      and (ret_uint = test_case[index].ret_uint)
		      and (ret_udint = test_case[index].ret_udint)
		      and (ret_real = test_case[index].ret_real)
		      and (ret_lreal = test_case[index].ret_lreal));

		(* ---------- log message ---------------*)
		expected := '';
		expected := CONCAT(expected, comma_blank, int_to_string(test_case[index].ret_int));
		expected := CONCAT(expected, comma_blank, dint_to_string(test_case[index].ret_dint));
		expected := CONCAT(expected, comma_blank, uint_to_string(test_case[index].ret_uint));
		expected := CONCAT(expected, comma_blank, udint_to_string(test_case[index].ret_udint));
		expected := CONCAT(expected, comma_blank, real_to_string(test_case[index].ret_real));
		expected := CONCAT(expected, comma_blank, lreal_to_string(test_case[index].ret_lreal));
		obtained := '';
		obtained := CONCAT(obtained, comma_blank, int_to_string(ret_int));
		obtained := CONCAT(obtained, comma_blank, dint_to_string(ret_dint));
		obtained := CONCAT(obtained, comma_blank, uint_to_string(ret_uint));
		obtained := CONCAT(obtained, comma_blank, udint_to_string(ret_udint));
		obtained := CONCAT(obtained, comma_blank, real_to_string(ret_real));
		obtained := CONCAT(obtained, comma_blank, lreal_to_string(ret_lreal));

		(* ---------- cycle ----------*)
		SingleTest(this, result, expected, obtained, test_cases,
				   index, test_level_18, test_counter_18, test_loops_18, test_errors_18);
	end_if;
END_PROGRAM

(* ---- add_sub_time_P.st ---- *)
(*[[ ]]*)
PROGRAM add_sub_time_P
#import "Crosstable.gvl"
#import "Resource1.gvl"
CONST
	this : int := 50;
	test_cases : int := 5;
END_CONST
VAR
	test_case : array [1..test_cases] of time2_time2_T := [
		(input0 := t#10ms, input1 := t#10ms, retval0 := t#20ms,  retval1 := t#0ms),
		(input0 := t#20ms, input1 := t#10ms, retval0 := t#30ms,  retval1 := t#10ms),
		(input0 := t#10s,  input1 := t#10s,  retval0 := t#20s,   retval1 := t#0s),
		(input0 := t#1s,   input1 := t#10ms, retval0 := t#1010ms,retval1 := t#990ms),
		(input0 := t#1s,   input1 := t#2s,   retval0 := t#3s,    retval1 := t#-1s)
	];
    retval0  : time;
    retval1  : time;

	index : int := 1;
	expected : string;
	obtained : string;
	result : bool;
END_VAR

	if Status = STATUS_RUNNING AND test_level_50 > TEST_DISABLED and test_loops_50 < Target then

		(* ---------- test action ---------------*)
        retval0     := add_time(test_case[index].input0, test_case[index].input1);
        retval1     := sub_time(test_case[index].input0, test_case[index].input1);

		(* ---------- test condition ---------------*)
        result := ((retval0 = test_case[index].retval0)
		       and (retval1 = test_case[index].retval1));

		(* ---------- log message ---------------*)
		expected := '';
		expected := CONCAT(expected, comma_blank, time_to_string(test_case[index].retval0));
		expected := CONCAT(expected, comma_blank, time_to_string(test_case[index].retval1));
		obtained := '';
		obtained := CONCAT(obtained, comma_blank, time_to_string(retval0));
		obtained := CONCAT(obtained, comma_blank, time_to_string(retval1));

		(* ---------- cycle ----------*)
		SingleTest(this, result, expected, obtained, test_cases,
				   index, test_level_50, test_counter_50, test_loops_50, test_errors_50);
	end_if;
END_PROGRAM

(* ---- and_P.st ---- *)
(*[[ ]]*)
PROGRAM and_P
#import "Crosstable.gvl"
#import "Resource1.gvl"
CONST
	this : int := 27;
	test_cases : int := 13;
END_CONST
VAR
	test_case : array [1..test_cases] of bit2_bit_T := [
		(input0 := 0, 		    input1 := 0, 	 	   ret_bool := 0, ret_byte := 0, 	 ret_word := 0, 	ret_dword := 0),
		(input0 := 0, 			input1 := 1, 	   	   ret_bool := 0, ret_byte := 0, 	 ret_word := 0, 	ret_dword := 0),
		(input0 := 1, 			input1 := 0, 	   	   ret_bool := 0, ret_byte := 0, 	 ret_word := 0, 	ret_dword := 0),
		(input0 := 1, 			input1 := 1, 	       ret_bool := 1, ret_byte := 1, 	 ret_word := 1, 	ret_dword := 1),
		(input0 := 0, 			input1 := 16#000000ff, ret_bool := 0, ret_byte := 0, 	 ret_word := 0, 	ret_dword := 0),
		(input0 := 16#000000ff, input1 := 16#000000ff, ret_bool := 1, ret_byte := 16#ff, ret_word := 16#00ff, ret_dword := 16#000000ff),
		(input0 := 16#0000000f, input1 := 16#000000f0, ret_bool := 1, ret_byte := 16#00, ret_word := 16#0000, ret_dword := 16#00000000),
		(input0 := 16#0000ffff, input1 := 16#0000ffff, ret_bool := 1, ret_byte := 16#ff, ret_word := 16#ffff, ret_dword := 16#0000ffff),
		(input0 := 16#0000ffff, input1 := 16#000000ff, ret_bool := 1, ret_byte := 16#ff, ret_word := 16#00ff, ret_dword := 16#000000ff),
		(input0 := 16#0000f000, input1 := 16#0000ffff, ret_bool := 1, ret_byte := 16#00, ret_word := 16#f000, ret_dword := 16#0000f000),
		(input0 := 16#000000ff, input1 := 16#0000ff00, ret_bool := 1, ret_byte := 16#00, ret_word := 16#0000, ret_dword := 16#00000000),
		(input0 := 16#abcde012, input1 := 16#ffffffff, ret_bool := 1, ret_byte := 16#12, ret_word := 16#e012, ret_dword := 16#abcde012),
		(input0 := 16#abcdefab, input1 := 16#ff000000, ret_bool := 1, ret_byte := 16#00, ret_word := 16#0000, ret_dword := 16#ab000000)
	];
    ret_bool   : bool;
    ret_byte   : byte;
    ret_word   : word;
    ret_dword  : dword;

	index : int := 1;
	expected : string;
	obtained : string;
	result : bool;
END_VAR

	if Status = STATUS_RUNNING AND test_level_27 > TEST_DISABLED and test_loops_27 < Target then

		(* ---------- test action ---------------*)
        ret_bool   := and(dword_to_bool(test_case[index].input0), dword_to_bool(test_case[index].input1));
        ret_byte   := and(dword_to_byte(test_case[index].input0), dword_to_byte(test_case[index].input1));
        ret_word   := and(dword_to_word(test_case[index].input0), dword_to_word(test_case[index].input1));
        ret_dword  := and(test_case[index].input0, test_case[index].input1);

		(* ---------- test condition ---------------*)
        result := (ret_bool = test_case[index].ret_bool)
		      and (ret_byte = test_case[index].ret_byte)
		      and (ret_word = test_case[index].ret_word)
		      and (ret_dword = test_case[index].ret_dword);

		(* ---------- log message ---------------*)
		expected := '';
		expected := CONCAT(expected, comma_blank, bool_to_string(test_case[index].ret_bool));
		expected := CONCAT(expected, comma_blank, byte_to_string(test_case[index].ret_byte));
		expected := CONCAT(expected, comma_blank, word_to_string(test_case[index].ret_word));
		expected := CONCAT(expected, comma_blank, dword_to_string(test_case[index].ret_dword));
		obtained := '';
		obtained := CONCAT(obtained, comma_blank, bool_to_string(ret_bool));
		obtained := CONCAT(obtained, comma_blank, byte_to_string(ret_byte));
		obtained := CONCAT(obtained, comma_blank, word_to_string(ret_word));
		obtained := CONCAT(obtained, comma_blank, dword_to_string(ret_dword));

		(* ---------- cycle ----------*)
		SingleTest(this, result, expected, obtained, test_cases,
				   index, test_level_27, test_counter_27, test_loops_27, test_errors_27);
	end_if;
END_PROGRAM

(* ---- bool_to_all_P.st ---- *)
(*[[ ]]*)
PROGRAM bool_to_all_P
#import "Crosstable.gvl"
#import "Resource1.gvl"
CONST
	this : int := 1;
	test_cases : int := 2;
END_CONST
VAR
	test_case : array [1..test_cases] of bool_all_T := [
		(input := false, ret_byte := 0, ret_dint := 0, ret_dword := 0, ret_int := 0, ret_lreal := 0.0, ret_real := 0.0,
		   ret_string := 'false', ret_udint := 0, ret_uint := 0, ret_word := 0),
		(input := true, ret_byte := 1, ret_dint := 1, ret_dword := 1, ret_int := 1, ret_lreal := 1.0, ret_real := 1.0,
		   ret_string := 'true', ret_udint := 1, ret_uint := 1, ret_word := 1)
	];
    ret_byte   : byte;
    ret_dint   : dint;
    ret_dword  : dword;
    ret_int    : int;
    ret_lreal  : lreal;
    ret_real   : real;
    ret_string : string;
    ret_udint  : udint;
    ret_uint   : uint;
    ret_word   : word;

	index : int := 1;
	expected : string;
	obtained : string;
	result : bool;
END_VAR

	if Status = STATUS_RUNNING AND test_level_01 > TEST_DISABLED and test_loops_01 < Target then

		(* ---------- test action ---------------*)
        ret_byte   := bool_to_byte(test_case[index].input);
        ret_dint   := bool_to_dint(test_case[index].input);
        ret_dword  := bool_to_dword(test_case[index].input);
        ret_int    := bool_to_int(test_case[index].input);
        ret_lreal  := bool_to_lreal(test_case[index].input);
        ret_real   := bool_to_real(test_case[index].input);
        ret_string := bool_to_string(test_case[index].input);
        ret_udint  := bool_to_udint(test_case[index].input);
        ret_uint   := bool_to_uint(test_case[index].input);
        ret_word   := bool_to_word(test_case[index].input);

		(* ---------- test condition ---------------*)
        result := (ret_byte = test_case[index].ret_byte)
		      and (ret_dint = test_case[index].ret_dint)
		      and (ret_dword = test_case[index].ret_dword)
		      and (ret_int = test_case[index].ret_int)
		      and (ret_lreal = test_case[index].ret_lreal)
		      and (ret_real = test_case[index].ret_real)
		      and (ret_string = test_case[index].ret_string)
		      and (ret_udint = test_case[index].ret_udint)
		      and (ret_uint = test_case[index].ret_uint)
		      and (ret_word = test_case[index].ret_word);

		(* ---------- log message ---------------*)
		expected := '';
		expected := CONCAT(expected, comma_blank, byte_to_string(test_case[index].ret_byte));
		expected := CONCAT(expected, comma_blank, dint_to_string(test_case[index].ret_dint));
		expected := CONCAT(expected, comma_blank, dword_to_string(test_case[index].ret_dword));
		expected := CONCAT(expected, comma_blank, int_to_string(test_case[index].ret_int));
		expected := CONCAT(expected, comma_blank, lreal_to_string(test_case[index].ret_lreal));
		expected := CONCAT(expected, comma_blank, real_to_string(test_case[index].ret_real));
		expected := CONCAT(expected, comma_blank, test_case[index].ret_string);
		expected := CONCAT(expected, comma_blank, udint_to_string(test_case[index].ret_udint));
		expected := CONCAT(expected, comma_blank, uint_to_string(test_case[index].ret_uint));
		expected := CONCAT(expected, comma_blank, word_to_string(test_case[index].ret_word));
		obtained := '';
		obtained := CONCAT(obtained, comma_blank, byte_to_string(ret_byte));
		obtained := CONCAT(obtained, comma_blank, dint_to_string(ret_dint));
		obtained := CONCAT(obtained, comma_blank, dword_to_string(ret_dword));
		obtained := CONCAT(obtained, comma_blank, int_to_string(ret_int));
		obtained := CONCAT(obtained, comma_blank, lreal_to_string(ret_lreal));
		obtained := CONCAT(obtained, comma_blank, real_to_string(ret_real));
		obtained := CONCAT(obtained, comma_blank, ret_string);
		obtained := CONCAT(obtained, comma_blank, udint_to_string(ret_udint));
		obtained := CONCAT(obtained, comma_blank, uint_to_string(ret_uint));
		obtained := CONCAT(obtained, comma_blank, word_to_string(ret_word));

		(* ---------- cycle ----------*)
		SingleTest(this, result, expected, obtained, test_cases,
				   index, test_level_01, test_counter_01, test_loops_01, test_errors_01);
	end_if;
END_PROGRAM

(* ---- byte_swap_P.st ---- *)
(*[[ ]]*)
PROGRAM byte_swap_P
#import "Crosstable.gvl"
#import "Resource1.gvl"
CONST
	this : int := 56;
	test_cases : int := 5;
END_CONST
VAR
	test_case : array [1..test_cases] of bit_bit_T := [
		(input := 0, 		   ret_word := 16#0000, ret_dword := 16#00000000),
		(input := 16#000000ff, ret_word := 16#ff00, ret_dword := 16#ff000000),
		(input := 16#11223344, ret_word := 16#4433, ret_dword := 16#44332211),
		(input := 16#0000ffff, ret_word := 16#ffff, ret_dword := 16#ffff0000),
		(input := 16#12131415, ret_word := 16#1514, ret_dword := 16#15141312)
	];
    ret_word   : word;
    ret_dword  : dword;

	index : int := 1;
	expected : string;
	obtained : string;
	result : bool;
END_VAR

	if Status = STATUS_RUNNING AND test_level_56 > TEST_DISABLED and test_loops_56 < Target then

		(* ---------- test action ---------------*)
        ret_word   := byte_swap_word(dword_to_word(test_case[index].input));
        ret_dword  := byte_swap_dword(test_case[index].input);

		(* ---------- test condition ---------------*)
        result := (ret_word = test_case[index].ret_word)
		      and (ret_dword = test_case[index].ret_dword);

		(* ---------- log message ---------------*)
		expected := '';
		expected := CONCAT(expected, comma_blank, word_to_string(test_case[index].ret_word));
		expected := CONCAT(expected, comma_blank, dword_to_string(test_case[index].ret_dword));
		obtained := '';
		obtained := CONCAT(obtained, comma_blank, word_to_string(ret_word));
		obtained := CONCAT(obtained, comma_blank, dword_to_string(ret_dword));

		(* ---------- cycle ----------*)
		SingleTest(this, result, expected, obtained, test_cases,
				   index, test_level_56, test_counter_56, test_loops_56, test_errors_56);
	end_if;
END_PROGRAM

(* ---- byte_to_all_P.st ---- *)
(*[[
]]*)
PROGRAM byte_to_all_P
#import "Crosstable.gvl"
#import "Resource1.gvl"
CONST
	this : int := 2;
	test_cases : int := 3;
END_CONST
VAR
	test_case : array [1..test_cases] of byte_all_T := [
		(input := 0, ret_bool := 0, ret_dint := 0, ret_dword := 0, ret_int := 0, ret_lreal := 0.0, ret_real := 0.0,
		   ret_string := '0', ret_udint := 0, ret_uint := 0, ret_word := 0),
		(input := 1, ret_bool := 1, ret_dint := 1, ret_dword := 1, ret_int := 1, ret_lreal := 1.0, ret_real := 1.0,
		   ret_string := '1', ret_udint := 1, ret_uint := 1, ret_word := 1),
		(input := 255, ret_bool := 1, ret_dint := 255, ret_dword := 255, ret_int := 255, ret_lreal := 255.0, ret_real := 255.0,
		   ret_string := '255', ret_udint := 255, ret_uint := 255, ret_word := 255)
	];
    ret_bool   : bool;
    ret_dint   : dint;
    ret_dword  : dword;
    ret_int    : int;
    ret_lreal  : lreal;
    ret_real   : real;
    ret_string : string;
    ret_udint  : udint;
    ret_uint   : uint;
    ret_word   : word;

	index : int := 1;
	expected : string;
	obtained : string;
	result : bool;
END_VAR

	if Status = STATUS_RUNNING AND test_level_02 > TEST_DISABLED and test_loops_02 < Target then

		(* ---------- test action ---------------*)
        ret_bool   := byte_to_bool(test_case[index].input);
        ret_dint   := byte_to_dint(test_case[index].input);
        ret_dword  := byte_to_dword(test_case[index].input);
        ret_int    := byte_to_int(test_case[index].input);
        ret_lreal  := byte_to_lreal(test_case[index].input);
        ret_real   := byte_to_real(test_case[index].input);
        ret_string := byte_to_string(test_case[index].input);
        ret_udint  := byte_to_udint(test_case[index].input);
        ret_uint   := byte_to_uint(test_case[index].input);
        ret_word   := byte_to_word(test_case[index].input);

		(* ---------- test condition ---------------*)
        result := (ret_bool = test_case[index].ret_bool)
		      and (ret_dint = test_case[index].ret_dint)
		      and (ret_dword = test_case[index].ret_dword)
		      and (ret_int = test_case[index].ret_int)
		      and (ret_lreal = test_case[index].ret_lreal)
		      and (ret_real = test_case[index].ret_real)
		      and (ret_string = test_case[index].ret_string)
		      and (ret_udint = test_case[index].ret_udint)
		      and (ret_uint = test_case[index].ret_uint)
		      and (ret_word = test_case[index].ret_word);

		(* ---------- log message ---------------*)
		expected := '';
		expected := CONCAT(expected, comma_blank, bool_to_string(test_case[index].ret_bool));
		expected := CONCAT(expected, comma_blank, dint_to_string(test_case[index].ret_dint));
		expected := CONCAT(expected, comma_blank, dword_to_string(test_case[index].ret_dword));
		expected := CONCAT(expected, comma_blank, int_to_string(test_case[index].ret_int));
		expected := CONCAT(expected, comma_blank, lreal_to_string(test_case[index].ret_lreal));
		expected := CONCAT(expected, comma_blank, real_to_string(test_case[index].ret_real));
		expected := CONCAT(expected, comma_blank, test_case[index].ret_string);
		expected := CONCAT(expected, comma_blank, udint_to_string(test_case[index].ret_udint));
		expected := CONCAT(expected, comma_blank, uint_to_string(test_case[index].ret_uint));
		expected := CONCAT(expected, comma_blank, word_to_string(test_case[index].ret_word));
		obtained := '';
		obtained := CONCAT(obtained, comma_blank, bool_to_string(ret_bool));
		obtained := CONCAT(obtained, comma_blank, dint_to_string(ret_dint));
		obtained := CONCAT(obtained, comma_blank, dword_to_string(ret_dword));
		obtained := CONCAT(obtained, comma_blank, int_to_string(ret_int));
		obtained := CONCAT(obtained, comma_blank, lreal_to_string(ret_lreal));
		obtained := CONCAT(obtained, comma_blank, real_to_string(ret_real));
		obtained := CONCAT(obtained, comma_blank, ret_string);
		obtained := CONCAT(obtained, comma_blank, udint_to_string(ret_udint));
		obtained := CONCAT(obtained, comma_blank, uint_to_string(ret_uint));
		obtained := CONCAT(obtained, comma_blank, word_to_string(ret_word));

		(* ---------- cycle ----------*)
		SingleTest(this, result, expected, obtained, test_cases,
				   index, test_level_02, test_counter_02, test_loops_02, test_errors_02);
	end_if;
END_PROGRAM

(* ---- concat_P.st ---- *)
(*[[
]]*)
PROGRAM concat_P
#import "Crosstable.gvl"
#import "Resource1.gvl"
CONST
	this : int := 42;
	test_cases : int := 3;
END_CONST
VAR
	test_case : array [1..test_cases] of string3_string_T := [
		(input0 := 'prima', input1 := '_seconda', input2 := '_terza',  retval := 'prima_seconda_terza'),
		(input0 := 'testa', input1 := '', input2 := '_coda',  retval := 'testa_coda'),
		(input0 := '', input1 := 'senza', input2 := '_testa', retval := 'senza_testa')
	];
    retval : string;

	index : int := 1;
	expected : string;
	obtained : string;
	result : bool;
END_VAR

	if Status = STATUS_RUNNING AND test_level_42 > TEST_DISABLED and test_loops_42 < Target then

		(* ---------- test action ---------------*)
        retval := concat(test_case[index].input0, test_case[index].input1, test_case[index].input2);

		(* ---------- test condition ---------------*)
        result := (retval = test_case[index].retval);

		(* ---------- log message ---------------*)
		expected := '';
		expected := CONCAT(expected, comma_blank, test_case[index].retval);
		obtained := '';
		obtained := CONCAT(obtained, comma_blank, retval);

		(* ---------- cycle ----------*)
		SingleTest(this, result, expected, obtained, test_cases,
				   index, test_level_42, test_counter_42, test_loops_42, test_errors_42);
	end_if;
END_PROGRAM

(* ---- copy_byte_array_P.st ---- *)
(*[[
]]*)
PROGRAM copy_byte_array_P
#import "Crosstable.gvl"
#import "Resource1.gvl"
CONST
	this : int := 57;
	test_cases : int := 5;
END_CONST
VAR
	test_case : array [1..test_cases] of all_T :=
[
(in_bool:=0, in_byte:=0,   in_dint:=0,      in_dword:=0,   in_int:=0,   in_lreal:=0.0,   in_real:=0.0,
  in_string:='',			in_time:=t#0s, in_word:=0),
(in_bool:=1, in_byte:=1,   in_dint:=1,      in_dword:=1,   in_int:=1,   in_lreal:=1.1,   in_real:=1.1,
  in_string:='1',			in_time:=t#1s, in_word:=1),
(in_bool:=0, in_byte:=255, in_dint:=254,    in_dword:=253, in_int:=252, in_lreal:=251.0, in_real:=250.0,
  in_string:='stringa',		in_time:=t#249s, in_word:=16#248),
(in_bool:=0, in_byte:=111, in_dint:=123456, in_dword:=16#abcdef01, in_int:=23871, in_lreal:=0.01, in_real:=0.02,
  in_string:='stringa_molto_ma_molto_lunga', in_time:=t#249s, in_word:=16#abcd),
(in_bool:=0, in_byte:=16#ff, in_dint:=102030, in_dword:=16#1b0def01, in_int:=2387, in_lreal:=1.01, in_real:=2.02,
  in_string:='stringa_veramente_molto_ma_molto_ma_molto_ma_molto_lunga', in_time:=t#249ms, in_word:=16#ffbb)
];

	ret_bool   : bool;
	ret_byte   : byte;
	ret_dint   : dint;
	ret_dword  : dword;
	ret_int    : int;
	ret_lreal  : lreal;
	ret_real   : real;
	ret_string : string;
	ret_time   : time;
	ret_word   : word;
	byte_array : array[0..800] of byte;

	pos   : dint;
	index : int := 1;
	expected : string;
	obtained : string;
	result : bool;
END_VAR

	if Status = STATUS_RUNNING AND test_level_57 > TEST_DISABLED and test_loops_57 < Target then

		(* ---------- test action ---------------*)
		pos := 1;
		copy_bool_to_byte_array (test_case[index].in_bool, pos, byte_array);
		copy_byte_to_byte_array (test_case[index].in_byte, pos, byte_array);
		copy_dint_to_byte_array (test_case[index].in_dint, pos, byte_array);
		copy_dword_to_byte_array (test_case[index].in_dword, pos, byte_array);
		copy_int_to_byte_array  (test_case[index].in_int, pos, byte_array);
		copy_lreal_to_byte_array (test_case[index].in_lreal, pos, byte_array);
		copy_real_to_byte_array (test_case[index].in_real, pos, byte_array);
		copy_time_to_byte_array (test_case[index].in_time, pos, byte_array);
		copy_word_to_byte_array (test_case[index].in_word, pos, byte_array);
		copy_string_to_byte_array (test_case[index].in_string, pos, byte_array);

		pos := 1;
		ret_bool   := copy_bool_from_byte_array (pos, byte_array);
		ret_byte   := copy_byte_from_byte_array (pos, byte_array);
		ret_dint   := copy_dint_from_byte_array (pos, byte_array);
		ret_dword  := copy_dword_from_byte_array(pos, byte_array);
		ret_int    := copy_int_from_byte_array  (pos, byte_array);
		ret_lreal  := copy_lreal_from_byte_array(pos, byte_array);
		ret_real   := copy_real_from_byte_array (pos, byte_array);
		ret_time   := copy_time_from_byte_array (pos, byte_array);
		ret_word   := copy_word_from_byte_array (pos, byte_array);
		ret_string := copy_string_from_byte_array(pos, byte_array);

		(* NOTA BENE: la copy_string_*_byte_array funziona bene solo se è l'ultima;
		   altrimenti le funzioni successive non funzionano *)

		(* ---------- test condition ---------------*)
		result := (ret_bool   = test_case[index].in_bool)
		      and (ret_byte   = test_case[index].in_byte)
		      and (ret_dint   = test_case[index].in_dint)
		      and (ret_dword  = test_case[index].in_dword)
		      and (ret_int    = test_case[index].in_int)
		      and (ret_lreal  = test_case[index].in_lreal)
		      and (ret_real   = test_case[index].in_real)
		      and (ret_string = test_case[index].in_string)
		      and (ret_time   = test_case[index].in_time)
		      and (ret_word   = test_case[index].in_word);

		(* ---------- log message ---------------*)
		expected := '';
		expected := CONCAT(expected, comma_blank, bool_to_string(test_case[index].in_bool));
		expected := CONCAT(expected, comma_blank, byte_to_string(test_case[index].in_byte));
		expected := CONCAT(expected, comma_blank, dint_to_string(test_case[index].in_dint));
		expected := CONCAT(expected, comma_blank, dword_to_string(test_case[index].in_dword));
		expected := CONCAT(expected, comma_blank, int_to_string(test_case[index].in_int));
		expected := CONCAT(expected, comma_blank, lreal_to_string(test_case[index].in_lreal));
		expected := CONCAT(expected, comma_blank, real_to_string(test_case[index].in_real));
		expected := CONCAT(expected, comma_blank, test_case[index].in_string);
		expected := CONCAT(expected, comma_blank, time_to_string(test_case[index].in_time));
		expected := CONCAT(expected, comma_blank, word_to_string(test_case[index].in_word));
		obtained := '';
		obtained := CONCAT(obtained, comma_blank, bool_to_string(ret_bool));
		obtained := CONCAT(obtained, comma_blank, byte_to_string(ret_byte));
		obtained := CONCAT(obtained, comma_blank, dint_to_string(ret_dint));
		obtained := CONCAT(obtained, comma_blank, dword_to_string(ret_dword));
		obtained := CONCAT(obtained, comma_blank, int_to_string(ret_int));
		obtained := CONCAT(obtained, comma_blank, lreal_to_string(ret_lreal));
		obtained := CONCAT(obtained, comma_blank, real_to_string(ret_real));
		obtained := CONCAT(obtained, comma_blank, ret_string);
		obtained := CONCAT(obtained, comma_blank, time_to_string(ret_time));
		obtained := CONCAT(obtained, comma_blank, word_to_string(ret_word));

		(* ---------- cycle ----------*)
		SingleTest(this, result, expected, obtained, test_cases,
				   index, test_level_57, test_counter_57, test_loops_57, test_errors_57);
	end_if;

END_PROGRAM

(* ---- ct_P.st ---- *)
(*[[
]]*)
PROGRAM ct_P
#import "Crosstable.gvl"
#import "Resource1.gvl"
CONST
	this : int := 54;
	test_cases : int := 12;
END_CONST
VAR
	test_case : array [1..test_cases] of bool2_bool_int2_T := [
		(input1 := false, input2 := true,  retval1 := false, retval2 := 3, retval3 := 0),
		(input1 := false, input2 := false, retval1 := false, retval2 := 3, retval3 := 0),
		(input1 := true,  input2 := false, retval1 := false, retval2 := 2, retval3 := 1),

		(input1 := false, input2 := false, retval1 := false, retval2 := 2, retval3 := 1),
		(input1 := true,  input2 := false, retval1 := false, retval2 := 1, retval3 := 2),
		(input1 := true,  input2 := false, retval1 := false, retval2 := 1, retval3 := 2),

		(input1 := false, input2 := false, retval1 := false, retval2 := 1, retval3 := 2),
		(input1 := true,  input2 := false, retval1 := true,  retval2 := 0, retval3 := 3),
		(input1 := true,  input2 := false, retval1 := true,  retval2 := 0, retval3 := 3),

		(input1 := false, input2 := true,  retval1 := false, retval2 := 3, retval3 := 0),
		(input1 := false, input2 := false, retval1 := false, retval2 := 3, retval3 := 0),
		(input1 := true,  input2 := false, retval1 := false, retval2 := 2, retval3 := 1)
	];
    retval1  : bool;
    retval1bis : bool;
    retval2  : int;
    retval3  : int;

	CTD_Inst : CTD;
	CTU_Inst : CTU;
	index : int := 1;
	expected : string;
	obtained : string;
	result : bool;
END_VAR

	if Status = STATUS_RUNNING AND test_level_54 > TEST_DISABLED and test_loops_54 < Target then

		(* ---------- test action ---------------*)
		CTD_Inst(
			CD := test_case[index].input1, LD := test_case[index].input2, PV := 3,
			Q => retval1, CV => retval2);
		CTU_Inst(
			CU := test_case[index].input1, R := test_case[index].input2, PV := 3,
			Q => retval1bis, CV => retval3);

		(* ---------- test condition ---------------*)
        result := (retval1 = test_case[index].retval1)
		      and (retval1bis = test_case[index].retval1)
		      and (retval2 = test_case[index].retval2)
			  and (retval3 = test_case[index].retval3);

		(* ---------- log message ---------------*)
		expected := '';
		expected := CONCAT(expected, comma_blank, bool_to_string(test_case[index].retval1));
		expected := CONCAT(expected, comma_blank, bool_to_string(test_case[index].retval1));
		expected := CONCAT(expected, comma_blank, int_to_string(test_case[index].retval2));
		expected := CONCAT(expected, comma_blank, int_to_string(test_case[index].retval3));
		obtained := '';
		obtained := CONCAT(obtained, comma_blank, bool_to_string(retval1));
		obtained := CONCAT(obtained, comma_blank, bool_to_string(retval1bis));
		obtained := CONCAT(obtained, comma_blank, int_to_string(retval2));
		obtained := CONCAT(obtained, comma_blank, int_to_string(retval3));

		(* ---------- cycle ----------*)
		SingleTest(this, result, expected, obtained, test_cases,
				   index, test_level_54, test_counter_54, test_loops_54, test_errors_54);
	end_if;
END_PROGRAM

(* ---- delete_P.st ---- *)
(*[[ ]]*)
PROGRAM delete_P
#import "Crosstable.gvl"
#import "Resource1.gvl"
CONST
	this : int := 43;
	test_cases : int := 4;
END_CONST
VAR
	test_case : array [1..test_cases] of string_int2_string_T := [
		(input0 := 'stringa_di_test', input1 := 3,  input2 := 8, retval := 'stringa_test'),
		(input0 := 'stringa_di_test', input1 := 11, input2 := 0, retval := 'test'),
		(input0 := 'stringa_di_test', input1 := 8,  input2 := 8, retval := 'stringa'),
		(input0 := 'stringa_di_test', input1 := 100, input2 := 8, retval := 'stringa')
	];
    retval0   : string;
    retval1   : string;

	index : int := 1;
	expected : string;
	obtained : string;
	result : bool;
END_VAR

	if Status = STATUS_RUNNING AND test_level_43 > TEST_DISABLED and test_loops_43 < Target then

		(* ---------- test action ---------------*)
        retval0 := delete(test_case[index].input0, test_case[index].input1, test_case[index].input2);
        retval1 := delete(test_case[index].input0, int_to_dint(test_case[index].input1), int_to_dint(test_case[index].input2));

		(* ---------- test condition ---------------*)
        result := (retval0 = test_case[index].retval)
		      and (retval1 = test_case[index].retval);

		(* ---------- log message ---------------*)
		expected := '';
		expected := CONCAT(expected, comma_blank, test_case[index].retval);
		expected := CONCAT(expected, comma_blank, test_case[index].retval);
		obtained := '';
		obtained := CONCAT(obtained, comma_blank, retval0);
		obtained := CONCAT(obtained, comma_blank, retval1);

		(* ---------- cycle ----------*)
		SingleTest(this, result, expected, obtained, test_cases,
				   index, test_level_43, test_counter_43, test_loops_43, test_errors_43);
	end_if;
END_PROGRAM

(* ---- dint_to_all_P.st ---- *)
(*[[
]]*)
PROGRAM dint_to_all_P
#import "Crosstable.gvl"
#import "Resource1.gvl"
CONST
	this : int := 3;
	test_cases : int := 5;
END_CONST
VAR
	test_case : array [1..test_cases] of dint_all_T := [
		(input := 0, ret_bool := 0, ret_byte := 0, ret_dword := 0, ret_int := 0, ret_lreal := 0.0, ret_real := 0.0,
		   ret_string := '0', ret_time := t#0ms, ret_udint := 0, ret_uint := 0, ret_word := 0),
		(input := 1, ret_bool := 1, ret_byte := 1, ret_dword := 1, ret_int := 1, ret_lreal := 1.0, ret_real := 1.0,
		   ret_string := '1', ret_time := t#1ms, ret_udint := 1, ret_uint := 1, ret_word := 1),
		(input := -1, ret_bool := 1, ret_byte := 255, ret_dword := 4294967295, ret_int := -1, ret_lreal := -1.0, ret_real := -1.0,
		   ret_string := '-1', ret_time := t#-1ms, ret_udint := 4294967295, ret_uint := 65535, ret_word := 65535),
		(input := 255, ret_bool := 1, ret_byte := 255, ret_dword := 255, ret_int := 255, ret_lreal := 255.0, ret_real := 255.0,
		   ret_string := '255', ret_time := t#255ms, ret_udint := 255, ret_uint := 255, ret_word := 255),
		(input := 400, ret_bool := 1, ret_byte := 144, ret_dword := 400, ret_int := 400, ret_lreal := 400.0, ret_real := 400.0,
		   ret_string := '400', ret_time := t#400ms, ret_udint := 400, ret_uint := 400, ret_word := 400)
	];
    ret_bool   : bool;
    ret_byte   : byte;
    ret_dword  : dword;
    ret_int    : int;
    ret_lreal  : lreal;
    ret_real   : real;
    ret_string : string;
    ret_time   : time;
    ret_udint  : udint;
    ret_uint   : uint;
    ret_word   : word;

	index : int := 1;
	expected : string;
	obtained : string;
	result : bool;
END_VAR

	if Status = STATUS_RUNNING AND test_level_03 > TEST_DISABLED and test_loops_03 < Target then

		(* ---------- test action ---------------*)
        ret_bool   := dint_to_bool(test_case[index].input);
        ret_byte   := dint_to_byte(test_case[index].input);
        ret_dword  := dint_to_dword(test_case[index].input);
        ret_int    := dint_to_int(test_case[index].input);
        ret_lreal  := dint_to_lreal(test_case[index].input);
        ret_real   := dint_to_real(test_case[index].input);
        ret_string := dint_to_string(test_case[index].input);
        ret_time   := dint_to_time(test_case[index].input);
        ret_udint  := dint_to_udint(test_case[index].input);
        ret_uint   := dint_to_uint(test_case[index].input);
        ret_word   := dint_to_word(test_case[index].input);

		(* ---------- test condition ---------------*)
        result := (ret_bool = test_case[index].ret_bool)
		      and (ret_byte = test_case[index].ret_byte)
		      and (ret_dword = test_case[index].ret_dword)
		      and (ret_int = test_case[index].ret_int)
		      and (ret_lreal = test_case[index].ret_lreal)
		      and (ret_real = test_case[index].ret_real)
		      and (ret_string = test_case[index].ret_string)
		      and (ret_time = test_case[index].ret_time)
		      and (ret_udint = test_case[index].ret_udint)
		      and (ret_uint = test_case[index].ret_uint)
		      and (ret_word = test_case[index].ret_word);

		(* ---------- log message ---------------*)
		expected := '';
		expected := CONCAT(expected, comma_blank, bool_to_string(test_case[index].ret_bool));
		expected := CONCAT(expected, comma_blank, byte_to_string(test_case[index].ret_byte));
		expected := CONCAT(expected, comma_blank, dword_to_string(test_case[index].ret_dword));
		expected := CONCAT(expected, comma_blank, int_to_string(test_case[index].ret_int));
		expected := CONCAT(expected, comma_blank, lreal_to_string(test_case[index].ret_lreal));
		expected := CONCAT(expected, comma_blank, real_to_string(test_case[index].ret_real));
		expected := CONCAT(expected, comma_blank, test_case[index].ret_string);
		expected := CONCAT(expected, comma_blank, time_to_string(test_case[index].ret_time));
		expected := CONCAT(expected, comma_blank, udint_to_string(test_case[index].ret_udint));
		expected := CONCAT(expected, comma_blank, uint_to_string(test_case[index].ret_uint));
		expected := CONCAT(expected, comma_blank, word_to_string(test_case[index].ret_word));
		obtained := '';
		obtained := CONCAT(obtained, comma_blank, bool_to_string(ret_bool));
		obtained := CONCAT(obtained, comma_blank, byte_to_string(ret_byte));
		obtained := CONCAT(obtained, comma_blank, dword_to_string(ret_dword));
		obtained := CONCAT(obtained, comma_blank, int_to_string(ret_int));
		obtained := CONCAT(obtained, comma_blank, lreal_to_string(ret_lreal));
		obtained := CONCAT(obtained, comma_blank, real_to_string(ret_real));
		obtained := CONCAT(obtained, comma_blank, ret_string);
		obtained := CONCAT(obtained, comma_blank, udint_to_string(ret_udint));
		obtained := CONCAT(obtained, comma_blank, time_to_string(ret_time));
		obtained := CONCAT(obtained, comma_blank, uint_to_string(ret_uint));
		obtained := CONCAT(obtained, comma_blank, word_to_string(ret_word));

		(* ---------- cycle ----------*)
		SingleTest(this, result, expected, obtained, test_cases,
				   index, test_level_03, test_counter_03, test_loops_03, test_errors_03);
	end_if;

END_PROGRAM

(* ---- div_mul_time_P.st ---- *)
(*[[ ]]*)
PROGRAM div_mul_time_P
#import "Crosstable.gvl"
#import "Resource1.gvl"
CONST
	this : int := 51;
	test_cases : int := 4;
END_CONST
VAR
	test_case : array [1..test_cases] of time_num_time2_T := [
		(input0 := t#10ms, input1 := 1.0, retval0 := t#10ms,  retval1 := t#10ms),
		(input0 := t#20ms, input1 := 2.0, retval0 := t#10ms,  retval1 := t#40ms),
		(input0 := t#10s,  input1 := 1.0, retval0 := t#10s,   retval1 := t#10s),
		(input0 := t#20s,  input1 := 2.0, retval0 := t#10s,   retval1 := t#40s)
	];
    retval0  : time;
    retval1  : time;
    retval2  : time;
    retval3  : time;
    retval4  : time;
    retval5  : time;
    retval6  : time;
    retval7  : time;

	index : int := 1;
	expected : string;
	obtained : string;
	result : bool;
END_VAR

	if Status = STATUS_RUNNING AND test_level_51 > TEST_DISABLED and test_loops_51 < Target then

		(* ---------- test action ---------------*)
        retval0   := divtime(test_case[index].input0, lreal_to_int(test_case[index].input1));
        retval1   := divtime(test_case[index].input0, lreal_to_dint(test_case[index].input1));
        retval2   := divtime(test_case[index].input0, lreal_to_real(test_case[index].input1));
        retval3   := divtime(test_case[index].input0, test_case[index].input1);

        retval4   := multime(test_case[index].input0, lreal_to_int(test_case[index].input1));
        retval5   := multime(test_case[index].input0, lreal_to_dint(test_case[index].input1));
        retval6   := multime(test_case[index].input0, lreal_to_real(test_case[index].input1));
        retval7   := multime(test_case[index].input0, test_case[index].input1);

		(* ---------- test condition ---------------*)
        result := ((retval0 = test_case[index].retval0)
		       and (retval1 = test_case[index].retval0)
		       and (retval2 = test_case[index].retval0)
		       and (retval3 = test_case[index].retval0)
			   and (retval4 = test_case[index].retval1)
			   and (retval5 = test_case[index].retval1)
			   and (retval6 = test_case[index].retval1)
			   and (retval7 = test_case[index].retval1));

		(* ---------- log message ---------------*)
		expected := '';
		expected := CONCAT(expected, comma_blank, time_to_string(test_case[index].retval0));
		expected := CONCAT(expected, comma_blank, time_to_string(test_case[index].retval0));
		expected := CONCAT(expected, comma_blank, time_to_string(test_case[index].retval0));
		expected := CONCAT(expected, comma_blank, time_to_string(test_case[index].retval0));
		expected := CONCAT(expected, comma_blank, time_to_string(test_case[index].retval1));
		expected := CONCAT(expected, comma_blank, time_to_string(test_case[index].retval1));
		expected := CONCAT(expected, comma_blank, time_to_string(test_case[index].retval1));
		expected := CONCAT(expected, comma_blank, time_to_string(test_case[index].retval1));
		obtained := '';
		obtained := CONCAT(obtained, comma_blank, time_to_string(retval0));
		obtained := CONCAT(obtained, comma_blank, time_to_string(retval1));
		obtained := CONCAT(obtained, comma_blank, time_to_string(retval2));
		obtained := CONCAT(obtained, comma_blank, time_to_string(retval3));
		obtained := CONCAT(obtained, comma_blank, time_to_string(retval4));
		obtained := CONCAT(obtained, comma_blank, time_to_string(retval5));
		obtained := CONCAT(obtained, comma_blank, time_to_string(retval6));
		obtained := CONCAT(obtained, comma_blank, time_to_string(retval7));

		(* ---------- cycle ----------*)
		SingleTest(this, result, expected, obtained, test_cases,
				   index, test_level_51, test_counter_51, test_loops_51, test_errors_51);
	end_if;
END_PROGRAM

(* ---- div_P.st ---- *)
(*[[ ]]*)
PROGRAM div_P
#import "Crosstable.gvl"
#import "Resource1.gvl"
CONST
	this : int := 19;
	test_cases : int := 4;
END_CONST
VAR
	test_case : array [1..test_cases] of num2_num_T := [
		(input0 := 40.0, input1 := 2.0, ret_int := 20, ret_dint := 20, ret_udint := 20, ret_uint := 20, ret_real := 20.0, ret_lreal := 20.0),
		(input0 := 110.0, input1 := 1.0, ret_int := 110, ret_dint := 110, ret_udint := 110, ret_uint := 110, ret_real := 110.0, ret_lreal := 110.0),
		(input0 := -10.0, input1 := 100.0, ret_int := 0, ret_dint := 0, ret_udint := 0, ret_uint := 0, ret_real := -0.1, ret_lreal := -0.1),
		(input0 := -1.0, input1 := -1.0, ret_int := 1, ret_dint := 1, ret_udint := 0, ret_uint := 0, ret_real := 1.0, ret_lreal := 1.0)
	];
    ret_int    : int;
    ret_dint   : dint;
    ret_uint   : uint;
    ret_udint  : udint;
    ret_real   : real;
    ret_lreal  : lreal;

	index : int := 1;
	expected : string;
	obtained : string;
	result : bool;
END_VAR

	if Status = STATUS_RUNNING AND test_level_19 > TEST_DISABLED and test_loops_19 < Target then

		(* ---------- test action ---------------*)
		(*[LIB_4CIEC1131_3_TABLE_24]: FATAL ERROR B0035: Division By Zero {POU:0x0015 Off:0x006e Inst:0x00eb}*)
        ret_int     := div(lreal_to_int(test_case[index].input0), lreal_to_int(test_case[index].input1));
        ret_dint    := div(lreal_to_dint(test_case[index].input0), lreal_to_dint(test_case[index].input1));
        ret_uint    := div(lreal_to_uint(test_case[index].input0), lreal_to_uint(ABS(test_case[index].input1)));
        ret_udint   := div(lreal_to_udint(test_case[index].input0), lreal_to_udint(ABS(test_case[index].input1)));
        ret_real    := div(lreal_to_real(test_case[index].input0), lreal_to_real(test_case[index].input1));
        ret_lreal   := div(test_case[index].input0, test_case[index].input1);

		(* ---------- test condition ---------------*)
        result := ((ret_int = test_case[index].ret_int)
		      and (ret_dint = test_case[index].ret_dint)
		      and (ret_uint = test_case[index].ret_uint)
		      and (ret_udint = test_case[index].ret_udint)
		      and (ret_real = test_case[index].ret_real)
		      and (ret_lreal = test_case[index].ret_lreal));

		(* ---------- log message ---------------*)
		expected := '';
		expected := CONCAT(expected, comma_blank, int_to_string(test_case[index].ret_int));
		expected := CONCAT(expected, comma_blank, dint_to_string(test_case[index].ret_dint));
		expected := CONCAT(expected, comma_blank, uint_to_string(test_case[index].ret_uint));
		expected := CONCAT(expected, comma_blank, udint_to_string(test_case[index].ret_udint));
		expected := CONCAT(expected, comma_blank, real_to_string(test_case[index].ret_real));
		expected := CONCAT(expected, comma_blank, lreal_to_string(test_case[index].ret_lreal));
		obtained := '';
		obtained := CONCAT(obtained, comma_blank, int_to_string(ret_int));
		obtained := CONCAT(obtained, comma_blank, dint_to_string(ret_dint));
		obtained := CONCAT(obtained, comma_blank, uint_to_string(ret_uint));
		obtained := CONCAT(obtained, comma_blank, udint_to_string(ret_udint));
		obtained := CONCAT(obtained, comma_blank, real_to_string(ret_real));
		obtained := CONCAT(obtained, comma_blank, lreal_to_string(ret_lreal));

		(* ---------- cycle ----------*)
		SingleTest(this, result, expected, obtained, test_cases,
				   index, test_level_19, test_counter_19, test_loops_19, test_errors_19);
	end_if;
END_PROGRAM

(* ---- dword_to_all_P.st ---- *)
(*[[
]]*)
PROGRAM dword_to_all_P
#import "Crosstable.gvl"
#import "Resource1.gvl"
CONST
	this : int := 4;
	test_cases : int := 4;
END_CONST
VAR
	test_case : array [1..test_cases] of dword_all_T := [
		(input := 0, ret_bool := 0, ret_byte := 0, ret_dint := 0, ret_int := 0, ret_lreal := 0.0, ret_real := 0.0,
		   ret_string := '0', ret_udint := 0, ret_uint := 0, ret_word := 0),
		(input := 1, ret_bool := 1, ret_byte := 1, ret_dint := 1, ret_int := 1, ret_lreal := 1.0, ret_real := 1.0,
		   ret_string := '1', ret_udint := 1, ret_uint := 1, ret_word := 1),
		(input := 255, ret_bool := 1, ret_byte := 255, ret_dint := 255, ret_int := 255, ret_lreal := 255.0, ret_real := 255.0,
		   ret_string := '255', ret_udint := 255, ret_uint := 255, ret_word := 255),
		(input := 400, ret_bool := 1, ret_byte := 144, ret_dint := 400, ret_int := 400, ret_lreal := 400.0, ret_real := 400.0,
		   ret_string := '400', ret_udint := 400, ret_uint := 400, ret_word := 400)
	];
    ret_bool   : bool;
    ret_byte   : byte;
    ret_dint   : dint;
    ret_int    : int;
    ret_lreal  : lreal;
    ret_real   : real;
    ret_string : string;
    ret_udint  : udint;
    ret_uint   : uint;
    ret_word   : word;

	index : int := 1;
	expected : string;
	obtained : string;
	result : bool;
END_VAR

	if Status = STATUS_RUNNING AND test_level_04 > TEST_DISABLED and test_loops_04 < Target then

		(* ---------- test action ---------------*)
        ret_bool   := dword_to_bool(test_case[index].input);
        ret_byte   := dword_to_byte(test_case[index].input);
        ret_dint   := dword_to_dint(test_case[index].input);
        ret_int    := dword_to_int(test_case[index].input);
        ret_lreal  := dword_to_lreal(test_case[index].input);
        ret_real   := dword_to_real(test_case[index].input);
        ret_string := dword_to_string(test_case[index].input);
        ret_udint  := dword_to_udint(test_case[index].input);
        ret_uint   := dword_to_uint(test_case[index].input);
        ret_word   := dword_to_word(test_case[index].input);

		(* ---------- test condition ---------------*)
        result := (ret_bool = test_case[index].ret_bool)
		      and (ret_byte = test_case[index].ret_byte)
		      and (ret_dint = test_case[index].ret_dint)
		      and (ret_int = test_case[index].ret_int)
		      and (ret_lreal = test_case[index].ret_lreal)
		      and (ret_real = test_case[index].ret_real)
		      and (ret_string = test_case[index].ret_string)
		      and (ret_udint = test_case[index].ret_udint)
		      and (ret_uint = test_case[index].ret_uint)
		      and (ret_word = test_case[index].ret_word);

		(* ---------- log message ---------------*)
		expected := '';
		expected := CONCAT(expected, comma_blank, bool_to_string(test_case[index].ret_bool));
		expected := CONCAT(expected, comma_blank, byte_to_string(test_case[index].ret_byte));
		expected := CONCAT(expected, comma_blank, dint_to_string(test_case[index].ret_dint));
		expected := CONCAT(expected, comma_blank, int_to_string(test_case[index].ret_int));
		expected := CONCAT(expected, comma_blank, lreal_to_string(test_case[index].ret_lreal));
		expected := CONCAT(expected, comma_blank, real_to_string(test_case[index].ret_real));
		expected := CONCAT(expected, comma_blank, test_case[index].ret_string);
		expected := CONCAT(expected, comma_blank, udint_to_string(test_case[index].ret_udint));
		expected := CONCAT(expected, comma_blank, uint_to_string(test_case[index].ret_uint));
		expected := CONCAT(expected, comma_blank, word_to_string(test_case[index].ret_word));
		obtained := '';
		obtained := CONCAT(obtained, comma_blank, bool_to_string(ret_bool));
		obtained := CONCAT(obtained, comma_blank, byte_to_string(ret_byte));
		obtained := CONCAT(obtained, comma_blank, dint_to_string(ret_dint));
		obtained := CONCAT(obtained, comma_blank, int_to_string(ret_int));
		obtained := CONCAT(obtained, comma_blank, lreal_to_string(ret_lreal));
		obtained := CONCAT(obtained, comma_blank, real_to_string(ret_real));
		obtained := CONCAT(obtained, comma_blank, ret_string);
		obtained := CONCAT(obtained, comma_blank, udint_to_string(ret_udint));
		obtained := CONCAT(obtained, comma_blank, uint_to_string(ret_uint));
		obtained := CONCAT(obtained, comma_blank, word_to_string(ret_word));

		(* ---------- cycle ----------*)
		SingleTest(this, result, expected, obtained, test_cases,
				   index, test_level_04, test_counter_04, test_loops_04, test_errors_04);
	end_if;

END_PROGRAM
